// TIA Portal V15.1 export
// export: Created 2024-06-21T08:41:20.379845Z, ExportSetting WithDefaults, DisplayName Totally Integrated Automation Portal, DisplayVersion V15.1 Update 5, DisplayName TIA Portal Openness, DisplayVersion V15.1 Update 5, DisplayName SINAMICS Startdrive Advanced, DisplayVersion V15.1, DisplayName G130, G150, S120, S150, SINAMICS MV, S210, DisplayVersion V15.1, DisplayName G110M, G120, G120C, G120D, G120P, DisplayVersion V15.1, DisplayName STEP 7 Professional, DisplayVersion V15.1 Update 5, DisplayName STEP 7 Safety, DisplayVersion V15.1, DisplayName WinCC Professional, DisplayVersion V15.1 Update 5, DisplayName SIMATIC Visualization Architect, DisplayVersion V15.1
FUNCTION_BLOCK "LGBCRClockStartStop"   // FB6679, FBD
TITLE = LGBCRClockStartStop
{ S7_Optimized_Access := 'TRUE' }
VERSION : 0.1
// stored: AutoNumber false, IsIECCheckEnabled false, IsRetainMemResEnabled false, MemoryReserve 100, SetENOAutomatically False, UDAEnableTagReadback false
   VAR_INPUT
      I_DBRecieve { ExternalAccessible := 'False'; ExternalVisible := 'False'; ExternalWritable := 'False'} : "SupervisionZM";   // Receive DB - Communication with control room
      C_EnableBreaks { ExternalAccessible := 'False'; ExternalVisible := 'False'; ExternalWritable := 'False'} : Bool;   // Enable Breaks
   END_VAR
   VAR_OUTPUT
      O_Start { ExternalAccessible := 'False'; ExternalVisible := 'False'; ExternalWritable := 'False'} : Bool;   // Start production line
      O_Stop { ExternalAccessible := 'False'; ExternalVisible := 'False'; ExternalWritable := 'False'} : Bool;   // Stop production line
      O_Break { ExternalAccessible := 'False'; ExternalVisible := 'False'; ExternalWritable := 'False'} : Bool;   // Break
      O_Rotation { ExternalAccessible := 'False'; ExternalVisible := 'False'; ExternalWritable := 'False'} : Bool;   // Rotation
      O_NbrActiveShift { ExternalAccessible := 'False'; ExternalVisible := 'False'; ExternalWritable := 'False'} : Int;   // Feedback to control room
      O_NbrActiveBreak { ExternalAccessible := 'False'; ExternalVisible := 'False'; ExternalWritable := 'False'} : Int;   // Feedback to control room
      O_AlarmABCondition { ExternalAccessible := 'False'; ExternalVisible := 'False'; ExternalWritable := 'False'} : Bool;   // Alarm AB Condition
      O_AlarmA { ExternalAccessible := 'False'; ExternalVisible := 'False'; ExternalWritable := 'False'} : Bool;   // Alarm A
      O_AlarmB { ExternalAccessible := 'False'; ExternalVisible := 'False'; ExternalWritable := 'False'} : Bool;   // Alarm B
      O_AlarmC { ExternalAccessible := 'False'; ExternalVisible := 'False'; ExternalWritable := 'False'} : Bool;   // Alarm C
      O_AlarmD { ExternalAccessible := 'False'; ExternalVisible := 'False'; ExternalWritable := 'False'} : Bool;   // Alarm D
      H_AlarmWord { ExternalAccessible := 'False'; ExternalVisible := 'False'; ExternalWritable := 'False'} : DWord;   // Alarmword for WinCC
   END_VAR
   VAR_IN_OUT
      IO_Modes : "Modes";   // Modes
      H_HMI : "H_HMI";   // Animation
      H_GBCRClockStartStop : "H_GBCRClockStartStop";   // Animation
   END_VAR
   VAR
      AD_SelForce { ExternalAccessible := 'False'; ExternalVisible := 'False'; ExternalWritable := 'False'} : Bool;   // FORCE is selected in control room
      AD_SelStop { ExternalAccessible := 'False'; ExternalVisible := 'False'; ExternalWritable := 'False'} : Bool;   // STOP is selected in control room
      AD_SelRelief { ExternalAccessible := 'False'; ExternalVisible := 'False'; ExternalWritable := 'False'} : Bool;   // RELIEF is selected in control room
      DateTimePlc { ExternalAccessible := 'False'; ExternalVisible := 'False'; ExternalWritable := 'False'} : Date_And_Time;   // Date and time from Plc
      ActualTimeOfDayPlc { ExternalAccessible := 'False'; ExternalVisible := 'False'; ExternalWritable := 'False'} : Time_Of_Day;   // Actual time of day calculated by PLC
      Shift01 { ExternalAccessible := 'False'; ExternalVisible := 'False'; ExternalWritable := 'False'} : Bool;   // Shift01 active
      Shift02 { ExternalAccessible := 'False'; ExternalVisible := 'False'; ExternalWritable := 'False'} : Bool;   // Shift02 active
      Shift03 { ExternalAccessible := 'False'; ExternalVisible := 'False'; ExternalWritable := 'False'} : Bool;   // Shift03 active
      Shift04 { ExternalAccessible := 'False'; ExternalVisible := 'False'; ExternalWritable := 'False'} : Bool;   // Shift04 active
      Shift05 { ExternalAccessible := 'False'; ExternalVisible := 'False'; ExternalWritable := 'False'} : Bool;   // Shift05 active
      Shift06 { ExternalAccessible := 'False'; ExternalVisible := 'False'; ExternalWritable := 'False'} : Bool;   // Shift06 active
      Break01 { ExternalAccessible := 'False'; ExternalVisible := 'False'; ExternalWritable := 'False'} : Bool;   // Break01 active
      Break02 { ExternalAccessible := 'False'; ExternalVisible := 'False'; ExternalWritable := 'False'} : Bool;   // Break02 active
      Break03 { ExternalAccessible := 'False'; ExternalVisible := 'False'; ExternalWritable := 'False'} : Bool;   // Break03 active
      Break04 { ExternalAccessible := 'False'; ExternalVisible := 'False'; ExternalWritable := 'False'} : Bool;   // Break04 active
      Break05 { ExternalAccessible := 'False'; ExternalVisible := 'False'; ExternalWritable := 'False'} : Bool;   // Break05 active
      Break06 { ExternalAccessible := 'False'; ExternalVisible := 'False'; ExternalWritable := 'False'} : Bool;   // Break06 active
      MorningShift_RotationTime01 { ExternalAccessible := 'False'; ExternalVisible := 'False'; ExternalWritable := 'False'} : Bool;   // Rotation active
      MorningShift_RotationTime02 { ExternalAccessible := 'False'; ExternalVisible := 'False'; ExternalWritable := 'False'} : Bool;   // Rotation active
      MorningShift_RotationTime03 { ExternalAccessible := 'False'; ExternalVisible := 'False'; ExternalWritable := 'False'} : Bool;   // Rotation active
      MorningShift_RotationTime04 { ExternalAccessible := 'False'; ExternalVisible := 'False'; ExternalWritable := 'False'} : Bool;   // Rotation active
      LateShift_RotationTime01 { ExternalAccessible := 'False'; ExternalVisible := 'False'; ExternalWritable := 'False'} : Bool;   // Rotation active
      LateShift_RotationTime02 { ExternalAccessible := 'False'; ExternalVisible := 'False'; ExternalWritable := 'False'} : Bool;   // Rotation active
      LateShift_RotationTime03 { ExternalAccessible := 'False'; ExternalVisible := 'False'; ExternalWritable := 'False'} : Bool;   // Rotation active
      LateShift_RotationTime04 { ExternalAccessible := 'False'; ExternalVisible := 'False'; ExternalWritable := 'False'} : Bool;   // Rotation active
      NightShift_RotationTime01 { ExternalAccessible := 'False'; ExternalVisible := 'False'; ExternalWritable := 'False'} : Bool;   // Rotation active
      NightShift_RotationTime02 { ExternalAccessible := 'False'; ExternalVisible := 'False'; ExternalWritable := 'False'} : Bool;   // Rotation active
      NightShift_RotationTime03 { ExternalAccessible := 'False'; ExternalVisible := 'False'; ExternalWritable := 'False'} : Bool;   // Rotation active
      NightShift_RotationTime04 { ExternalAccessible := 'False'; ExternalVisible := 'False'; ExternalWritable := 'False'} : Bool;   // Rotation active
      MorningShiftDay5_RotationTime01 { ExternalAccessible := 'False'; ExternalVisible := 'False'; ExternalWritable := 'False'} : Bool;   // Rotation active
      MorningShiftDay5_RotationTime02 { ExternalAccessible := 'False'; ExternalVisible := 'False'; ExternalWritable := 'False'} : Bool;   // Rotation active
      MorningShiftDay5_RotationTime03 { ExternalAccessible := 'False'; ExternalVisible := 'False'; ExternalWritable := 'False'} : Bool;   // Rotation active
      MorningShiftDay5_RotationTime04 { ExternalAccessible := 'False'; ExternalVisible := 'False'; ExternalWritable := 'False'} : Bool;   // Rotation active
      LateShiftDay5_RotationTime01 { ExternalAccessible := 'False'; ExternalVisible := 'False'; ExternalWritable := 'False'} : Bool;   // Rotation active
      LateShiftDay5_RotationTime02 { ExternalAccessible := 'False'; ExternalVisible := 'False'; ExternalWritable := 'False'} : Bool;   // Rotation active
      LateShiftDay5_RotationTime03 { ExternalAccessible := 'False'; ExternalVisible := 'False'; ExternalWritable := 'False'} : Bool;   // Rotation active
      LateShiftDay5_RotationTime04 { ExternalAccessible := 'False'; ExternalVisible := 'False'; ExternalWritable := 'False'} : Bool;   // Rotation active
      NightShiftDay5_RotationTime01 { ExternalAccessible := 'False'; ExternalVisible := 'False'; ExternalWritable := 'False'} : Bool;   // Rotation active
      NightShiftDay5_RotationTime02 { ExternalAccessible := 'False'; ExternalVisible := 'False'; ExternalWritable := 'False'} : Bool;   // Rotation active
      NightShiftDay5_RotationTime03 { ExternalAccessible := 'False'; ExternalVisible := 'False'; ExternalWritable := 'False'} : Bool;   // Rotation active
      NightShiftDay5_RotationTime04 { ExternalAccessible := 'False'; ExternalVisible := 'False'; ExternalWritable := 'False'} : Bool;   // Rotation active
      ShiftActive { ExternalAccessible := 'False'; ExternalVisible := 'False'; ExternalWritable := 'False'} : Bool;   // Shift active
      BreakActive { ExternalAccessible := 'False'; ExternalVisible := 'False'; ExternalWritable := 'False'} : Bool;   // Break active
      RotationActive { ExternalAccessible := 'False'; ExternalVisible := 'False'; ExternalWritable := 'False'} : Bool;   // Rotation active
      Production { ExternalAccessible := 'False'; ExternalVisible := 'False'; ExternalWritable := 'False'} : Bool;   // In production, production line can RUN
      Start { ExternalAccessible := 'False'; ExternalVisible := 'False'; ExternalWritable := 'False'} : Bool;   // Start production line
      Stop { ExternalAccessible := 'False'; ExternalVisible := 'False'; ExternalWritable := 'False'} : Bool;   // Stop production line
      NbrActiveShift { ExternalAccessible := 'False'; ExternalVisible := 'False'; ExternalWritable := 'False'} : Int;   // Feedback to control room
      NbrActiveBreak { ExternalAccessible := 'False'; ExternalVisible := 'False'; ExternalWritable := 'False'} : Int;   // Feedback to control room
      AlarmA { ExternalAccessible := 'False'; ExternalVisible := 'False'; ExternalWritable := 'False'} : Bool;   // Alarm A
      AlarmB { ExternalAccessible := 'False'; ExternalVisible := 'False'; ExternalWritable := 'False'} : Bool;   // Alarm B
      AlarmC { ExternalAccessible := 'False'; ExternalVisible := 'False'; ExternalWritable := 'False'} : Bool;   // Alarm C
      AlarmD { ExternalAccessible := 'False'; ExternalVisible := 'False'; ExternalWritable := 'False'} : Bool;   // Alarm D
      AlarmABCondition { ExternalAccessible := 'False'; ExternalVisible := 'False'; ExternalWritable := 'False'} : Bool;   // Alarm AB Condition
      RotationTime { ExternalAccessible := 'False'; ExternalVisible := 'False'; ExternalWritable := 'False'} : Time_Of_Day;   // Rotation Time
      MorningShift_RotationTime01_End { ExternalAccessible := 'False'; ExternalVisible := 'False'; ExternalWritable := 'False'} : Time_Of_Day;   // Rotation End Time
      MorningShift_RotationTime02_End { ExternalAccessible := 'False'; ExternalVisible := 'False'; ExternalWritable := 'False'} : Time_Of_Day;   // Rotation End Time
      MorningShift_RotationTime03_End { ExternalAccessible := 'False'; ExternalVisible := 'False'; ExternalWritable := 'False'} : Time_Of_Day;   // Rotation End Time
      MorningShift_RotationTime04_End { ExternalAccessible := 'False'; ExternalVisible := 'False'; ExternalWritable := 'False'} : Time_Of_Day;   // Rotation End Time
      LateShift_RotationTime01_End { ExternalAccessible := 'False'; ExternalVisible := 'False'; ExternalWritable := 'False'} : Time_Of_Day;   // Rotation End Time
      LateShift_RotationTime02_End { ExternalAccessible := 'False'; ExternalVisible := 'False'; ExternalWritable := 'False'} : Time_Of_Day;   // Rotation End Time
      LateShift_RotationTime03_End { ExternalAccessible := 'False'; ExternalVisible := 'False'; ExternalWritable := 'False'} : Time_Of_Day;   // Rotation End Time
      LateShift_RotationTime04_End { ExternalAccessible := 'False'; ExternalVisible := 'False'; ExternalWritable := 'False'} : Time_Of_Day;   // Rotation End Time
      NightShift_RotationTime01_End { ExternalAccessible := 'False'; ExternalVisible := 'False'; ExternalWritable := 'False'} : Time_Of_Day;   // Rotation End Time
      NightShift_RotationTime02_End { ExternalAccessible := 'False'; ExternalVisible := 'False'; ExternalWritable := 'False'} : Time_Of_Day;   // Rotation End Time
      NightShift_RotationTime03_End { ExternalAccessible := 'False'; ExternalVisible := 'False'; ExternalWritable := 'False'} : Time_Of_Day;   // Rotation End Time
      NightShift_RotationTime04_End { ExternalAccessible := 'False'; ExternalVisible := 'False'; ExternalWritable := 'False'} : Time_Of_Day;   // Rotation End Time
      MorningShiftDay5_RotationTime01_End { ExternalAccessible := 'False'; ExternalVisible := 'False'; ExternalWritable := 'False'} : Time_Of_Day;   // Rotation End Time
      MorningShiftDay5_RotationTime02_End { ExternalAccessible := 'False'; ExternalVisible := 'False'; ExternalWritable := 'False'} : Time_Of_Day;   // Rotation End Time
      MorningShiftDay5_RotationTime03_End { ExternalAccessible := 'False'; ExternalVisible := 'False'; ExternalWritable := 'False'} : Time_Of_Day;   // Rotation End Time
      MorningShiftDay5_RotationTime04_End { ExternalAccessible := 'False'; ExternalVisible := 'False'; ExternalWritable := 'False'} : Time_Of_Day;   // Rotation End Time
      LateShiftDay5_RotationTime01_End { ExternalAccessible := 'False'; ExternalVisible := 'False'; ExternalWritable := 'False'} : Time_Of_Day;   // Rotation End Time
      LateShiftDay5_RotationTime02_End { ExternalAccessible := 'False'; ExternalVisible := 'False'; ExternalWritable := 'False'} : Time_Of_Day;   // Rotation End Time
      LateShiftDay5_RotationTime03_End { ExternalAccessible := 'False'; ExternalVisible := 'False'; ExternalWritable := 'False'} : Time_Of_Day;   // Rotation End Time
      LateShiftDay5_RotationTime04_End { ExternalAccessible := 'False'; ExternalVisible := 'False'; ExternalWritable := 'False'} : Time_Of_Day;   // Rotation End Time
      NightShiftDay5_RotationTime01_End { ExternalAccessible := 'False'; ExternalVisible := 'False'; ExternalWritable := 'False'} : Time_Of_Day;   // Rotation End Time
      NightShiftDay5_RotationTime02_End { ExternalAccessible := 'False'; ExternalVisible := 'False'; ExternalWritable := 'False'} : Time_Of_Day;   // Rotation End Time
      NightShiftDay5_RotationTime03_End { ExternalAccessible := 'False'; ExternalVisible := 'False'; ExternalWritable := 'False'} : Time_Of_Day;   // Rotation End Time
      NightShiftDay5_RotationTime04_End { ExternalAccessible := 'False'; ExternalVisible := 'False'; ExternalWritable := 'False'} : Time_Of_Day;   // Rotation End Time
      HMICmdCR { ExternalAccessible := 'False'; ExternalVisible := 'False'; ExternalWritable := 'False'} : Struct   // Temp / HMI Commands control room
         SelForce { ExternalAccessible := 'False'; ExternalVisible := 'False'; ExternalWritable := 'False'} : Bool;   // FORCE is selected in control room
         SelStop { ExternalAccessible := 'False'; ExternalVisible := 'False'; ExternalWritable := 'False'} : Bool;   // STOP is selected in control room
         SelRelief { ExternalAccessible := 'False'; ExternalVisible := 'False'; ExternalWritable := 'False'} : Bool;   // RELIEF is selected in control room
         Spare3 { ExternalAccessible := 'False'; ExternalVisible := 'False'; ExternalWritable := 'False'} : Bool;   // Spare
         Spare4 { ExternalAccessible := 'False'; ExternalVisible := 'False'; ExternalWritable := 'False'} : Bool;   // Spare
         Spare5 { ExternalAccessible := 'False'; ExternalVisible := 'False'; ExternalWritable := 'False'} : Bool;   // Spare
         Spare6 { ExternalAccessible := 'False'; ExternalVisible := 'False'; ExternalWritable := 'False'} : Bool;   // Spare
         Spare7 { ExternalAccessible := 'False'; ExternalVisible := 'False'; ExternalWritable := 'False'} : Bool;   // Spare
         Spare8 { ExternalAccessible := 'False'; ExternalVisible := 'False'; ExternalWritable := 'False'} : Bool;   // Spare
         Spare9 { ExternalAccessible := 'False'; ExternalVisible := 'False'; ExternalWritable := 'False'} : Bool;   // Spare
         Spare10 { ExternalAccessible := 'False'; ExternalVisible := 'False'; ExternalWritable := 'False'} : Bool;   // Spare
         Spare11 { ExternalAccessible := 'False'; ExternalVisible := 'False'; ExternalWritable := 'False'} : Bool;   // Spare
         Spare12 { ExternalAccessible := 'False'; ExternalVisible := 'False'; ExternalWritable := 'False'} : Bool;   // Spare
         Spare13 { ExternalAccessible := 'False'; ExternalVisible := 'False'; ExternalWritable := 'False'} : Bool;   // Spare
         Spare14 { ExternalAccessible := 'False'; ExternalVisible := 'False'; ExternalWritable := 'False'} : Bool;   // Spare
         Spare15 { ExternalAccessible := 'False'; ExternalVisible := 'False'; ExternalWritable := 'False'} : Bool;   // Spare
         Spare16 { ExternalAccessible := 'False'; ExternalVisible := 'False'; ExternalWritable := 'False'} : Bool;   // Spare
         Spare17 { ExternalAccessible := 'False'; ExternalVisible := 'False'; ExternalWritable := 'False'} : Bool;   // Spare
         Spare18 { ExternalAccessible := 'False'; ExternalVisible := 'False'; ExternalWritable := 'False'} : Bool;   // Spare
         Spare19 { ExternalAccessible := 'False'; ExternalVisible := 'False'; ExternalWritable := 'False'} : Bool;   // Spare
         Spare20 { ExternalAccessible := 'False'; ExternalVisible := 'False'; ExternalWritable := 'False'} : Bool;   // Spare
         Spare21 { ExternalAccessible := 'False'; ExternalVisible := 'False'; ExternalWritable := 'False'} : Bool;   // Spare
         Spare22 { ExternalAccessible := 'False'; ExternalVisible := 'False'; ExternalWritable := 'False'} : Bool;   // Spare
         Spare23 { ExternalAccessible := 'False'; ExternalVisible := 'False'; ExternalWritable := 'False'} : Bool;   // Spare
         Spare24 { ExternalAccessible := 'False'; ExternalVisible := 'False'; ExternalWritable := 'False'} : Bool;   // Spare
         Spare25 { ExternalAccessible := 'False'; ExternalVisible := 'False'; ExternalWritable := 'False'} : Bool;   // Spare
         Spare26 { ExternalAccessible := 'False'; ExternalVisible := 'False'; ExternalWritable := 'False'} : Bool;   // Spare
         Spare27 { ExternalAccessible := 'False'; ExternalVisible := 'False'; ExternalWritable := 'False'} : Bool;   // Spare
         Spare28 { ExternalAccessible := 'False'; ExternalVisible := 'False'; ExternalWritable := 'False'} : Bool;   // Spare
         Spare29 { ExternalAccessible := 'False'; ExternalVisible := 'False'; ExternalWritable := 'False'} : Bool;   // Spare
         Spare30 { ExternalAccessible := 'False'; ExternalVisible := 'False'; ExternalWritable := 'False'} : Bool;   // Spare
         Spare31 { ExternalAccessible := 'False'; ExternalVisible := 'False'; ExternalWritable := 'False'} : Bool;   // Spare
      END_STRUCT;
      HMICmd { ExternalAccessible := 'False'; ExternalVisible := 'False'; ExternalWritable := 'False'} : Struct   // HMI Commands
         MorningShift_RotationTime01_Active { ExternalAccessible := 'False'; ExternalVisible := 'False'; ExternalWritable := 'False'} : Bool;   // Rotation time active
         MorningShift_RotationTime02_Active { ExternalAccessible := 'False'; ExternalVisible := 'False'; ExternalWritable := 'False'} : Bool;   // Rotation time active
         MorningShift_RotationTime03_Active { ExternalAccessible := 'False'; ExternalVisible := 'False'; ExternalWritable := 'False'} : Bool;   // Rotation time active
         MorningShift_RotationTime04_Active { ExternalAccessible := 'False'; ExternalVisible := 'False'; ExternalWritable := 'False'} : Bool;   // Rotation time active
         LateShift_RotationTime01_Active { ExternalAccessible := 'False'; ExternalVisible := 'False'; ExternalWritable := 'False'} : Bool;   // Rotation time active
         LateShift_RotationTime02_Active { ExternalAccessible := 'False'; ExternalVisible := 'False'; ExternalWritable := 'False'} : Bool;   // Rotation time active
         LateShift_RotationTime03_Active { ExternalAccessible := 'False'; ExternalVisible := 'False'; ExternalWritable := 'False'} : Bool;   // Rotation time active
         LateShift_RotationTime04_Active { ExternalAccessible := 'False'; ExternalVisible := 'False'; ExternalWritable := 'False'} : Bool;   // Rotation time active
         NightShift_RotationTime01_Active { ExternalAccessible := 'False'; ExternalVisible := 'False'; ExternalWritable := 'False'} : Bool;   // Rotation time active
         NightShift_RotationTime02_Active { ExternalAccessible := 'False'; ExternalVisible := 'False'; ExternalWritable := 'False'} : Bool;   // Rotation time active
         NightShift_RotationTime03_Active { ExternalAccessible := 'False'; ExternalVisible := 'False'; ExternalWritable := 'False'} : Bool;   // Rotation time active
         NightShift_RotationTime04_Active { ExternalAccessible := 'False'; ExternalVisible := 'False'; ExternalWritable := 'False'} : Bool;   // Rotation time active
         MorningShiftDay5_RotationTime01_Active { ExternalAccessible := 'False'; ExternalVisible := 'False'; ExternalWritable := 'False'} : Bool;   // Rotation time active
         MorningShiftDay5_RotationTime02_Active { ExternalAccessible := 'False'; ExternalVisible := 'False'; ExternalWritable := 'False'} : Bool;   // Rotation time active
         MorningShiftDay5_RotationTime03_Active { ExternalAccessible := 'False'; ExternalVisible := 'False'; ExternalWritable := 'False'} : Bool;   // Rotation time active
         MorningShiftDay5_RotationTime04_Active { ExternalAccessible := 'False'; ExternalVisible := 'False'; ExternalWritable := 'False'} : Bool;   // Rotation time active
         LateShiftDay5_RotationTime01_Active { ExternalAccessible := 'False'; ExternalVisible := 'False'; ExternalWritable := 'False'} : Bool;   // Rotation time active
         LateShiftDay5_RotationTime02_Active { ExternalAccessible := 'False'; ExternalVisible := 'False'; ExternalWritable := 'False'} : Bool;   // Rotation time active
         LateShiftDay5_RotationTime03_Active { ExternalAccessible := 'False'; ExternalVisible := 'False'; ExternalWritable := 'False'} : Bool;   // Rotation time active
         LateShiftDay5_RotationTime04_Active { ExternalAccessible := 'False'; ExternalVisible := 'False'; ExternalWritable := 'False'} : Bool;   // Rotation time active
         NightShiftDay5_RotationTime01_Active { ExternalAccessible := 'False'; ExternalVisible := 'False'; ExternalWritable := 'False'} : Bool;   // Rotation time active
         NightShiftDay5_RotationTime02_Active { ExternalAccessible := 'False'; ExternalVisible := 'False'; ExternalWritable := 'False'} : Bool;   // Rotation time active
         NightShiftDay5_RotationTime03_Active { ExternalAccessible := 'False'; ExternalVisible := 'False'; ExternalWritable := 'False'} : Bool;   // Rotation time active
         NightShiftDay5_RotationTime04_Active { ExternalAccessible := 'False'; ExternalVisible := 'False'; ExternalWritable := 'False'} : Bool;   // Rotation time active
      END_STRUCT;
   END_VAR
   VAR_TEMP
      TReadStatus : Int;   // Integer used store the status of the clock read
      TempTime : Time_Of_Day;
   END_VAR
   VAR_TEMP   // added for the SCL form of the ladder/FBD networks
      _w1 : Bool;
   END_VAR
BEGIN

REGION Network 1: **** 1 - Inputs **** HMI Commands / **** 1 - Inputs **** HMI Commands !!! Control room !!!
   // HMI Commands
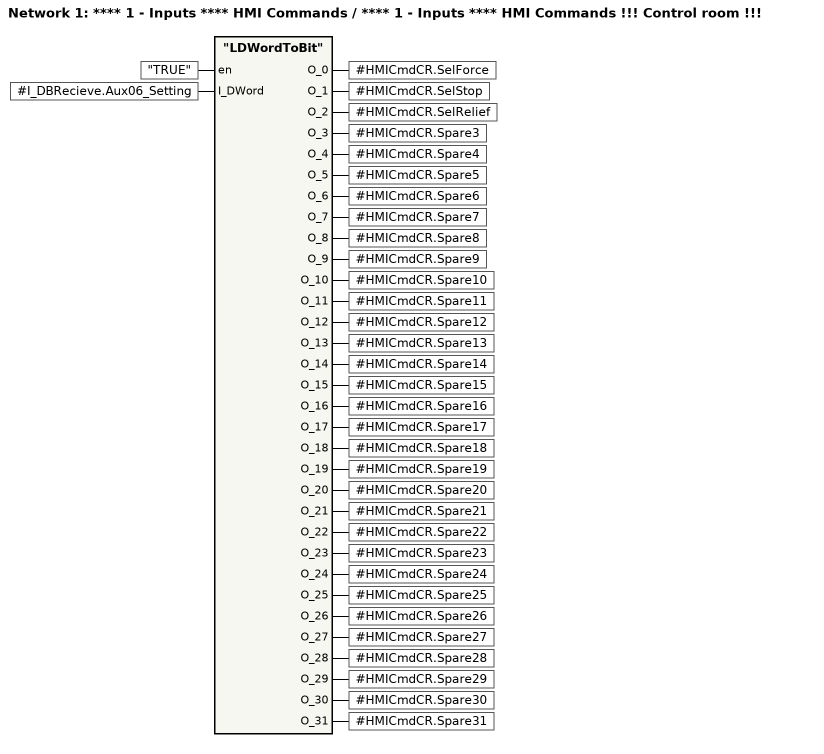
   IF "TRUE" THEN
       "LDWordToBit"(I_DWord := #I_DBRecieve.Aux06_Setting,
                     O_0 => #HMICmdCR.SelForce,
                     O_1 => #HMICmdCR.SelStop,
                     O_2 => #HMICmdCR.SelRelief,
                     O_3 => #HMICmdCR.Spare3,
                     O_4 => #HMICmdCR.Spare4,
                     O_5 => #HMICmdCR.Spare5,
                     O_6 => #HMICmdCR.Spare6,
                     O_7 => #HMICmdCR.Spare7,
                     O_8 => #HMICmdCR.Spare8,
                     O_9 => #HMICmdCR.Spare9,
                     O_10 => #HMICmdCR.Spare10,
                     O_11 => #HMICmdCR.Spare11,
                     O_12 => #HMICmdCR.Spare12,
                     O_13 => #HMICmdCR.Spare13,
                     O_14 => #HMICmdCR.Spare14,
                     O_15 => #HMICmdCR.Spare15,
                     O_16 => #HMICmdCR.Spare16,
                     O_17 => #HMICmdCR.Spare17,
                     O_18 => #HMICmdCR.Spare18,
                     O_19 => #HMICmdCR.Spare19,
                     O_20 => #HMICmdCR.Spare20,
                     O_21 => #HMICmdCR.Spare21,
                     O_22 => #HMICmdCR.Spare22,
                     O_23 => #HMICmdCR.Spare23,
                     O_24 => #HMICmdCR.Spare24,
                     O_25 => #HMICmdCR.Spare25,
                     O_26 => #HMICmdCR.Spare26,
                     O_27 => #HMICmdCR.Spare27,
                     O_28 => #HMICmdCR.Spare28,
                     O_29 => #HMICmdCR.Spare29,
                     O_30 => #HMICmdCR.Spare30,
                     O_31 => #HMICmdCR.Spare31);
   END_IF;
END_REGION

REGION Network 2: **** 1 - Inputs **** HMI Commands
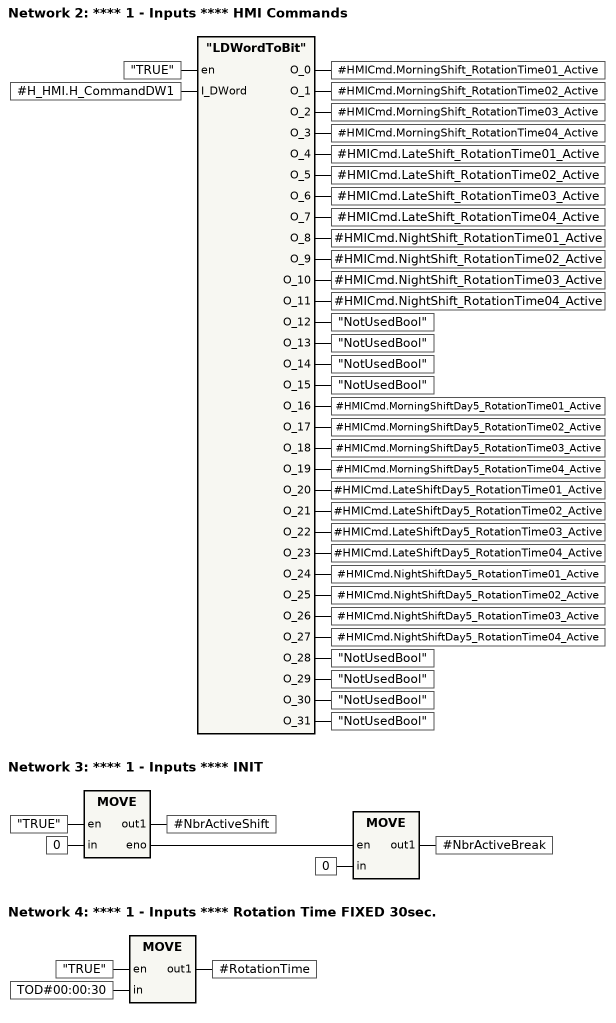
   IF "TRUE" THEN
       "LDWordToBit"(I_DWord := #H_HMI.H_CommandDW1,
                     O_0 => #HMICmd.MorningShift_RotationTime01_Active,
                     O_1 => #HMICmd.MorningShift_RotationTime02_Active,
                     O_2 => #HMICmd.MorningShift_RotationTime03_Active,
                     O_3 => #HMICmd.MorningShift_RotationTime04_Active,
                     O_4 => #HMICmd.LateShift_RotationTime01_Active,
                     O_5 => #HMICmd.LateShift_RotationTime02_Active,
                     O_6 => #HMICmd.LateShift_RotationTime03_Active,
                     O_7 => #HMICmd.LateShift_RotationTime04_Active,
                     O_8 => #HMICmd.NightShift_RotationTime01_Active,
                     O_9 => #HMICmd.NightShift_RotationTime02_Active,
                     O_10 => #HMICmd.NightShift_RotationTime03_Active,
                     O_11 => #HMICmd.NightShift_RotationTime04_Active,
                     O_12 => "NotUsedBool",
                     O_13 => "NotUsedBool",
                     O_14 => "NotUsedBool",
                     O_15 => "NotUsedBool",
                     O_16 => #HMICmd.MorningShiftDay5_RotationTime01_Active,
                     O_17 => #HMICmd.MorningShiftDay5_RotationTime02_Active,
                     O_18 => #HMICmd.MorningShiftDay5_RotationTime03_Active,
                     O_19 => #HMICmd.MorningShiftDay5_RotationTime04_Active,
                     O_20 => #HMICmd.LateShiftDay5_RotationTime01_Active,
                     O_21 => #HMICmd.LateShiftDay5_RotationTime02_Active,
                     O_22 => #HMICmd.LateShiftDay5_RotationTime03_Active,
                     O_23 => #HMICmd.LateShiftDay5_RotationTime04_Active,
                     O_24 => #HMICmd.NightShiftDay5_RotationTime01_Active,
                     O_25 => #HMICmd.NightShiftDay5_RotationTime02_Active,
                     O_26 => #HMICmd.NightShiftDay5_RotationTime03_Active,
                     O_27 => #HMICmd.NightShiftDay5_RotationTime04_Active,
                     O_28 => "NotUsedBool",
                     O_29 => "NotUsedBool",
                     O_30 => "NotUsedBool",
                     O_31 => "NotUsedBool");
   END_IF;
END_REGION

REGION Network 3: **** 1 - Inputs **** INIT
   IF "TRUE" THEN
       #NbrActiveShift := 0;
       #NbrActiveBreak := 0;
   END_IF;
END_REGION

REGION Network 4: **** 1 - Inputs **** Rotation Time FIXED 30sec.
   IF "TRUE" THEN #RotationTime := TOD#00:00:30; END_IF;
END_REGION

REGION Network 5: **** 1 - Inputs **** Rotation End Time Morning Shift
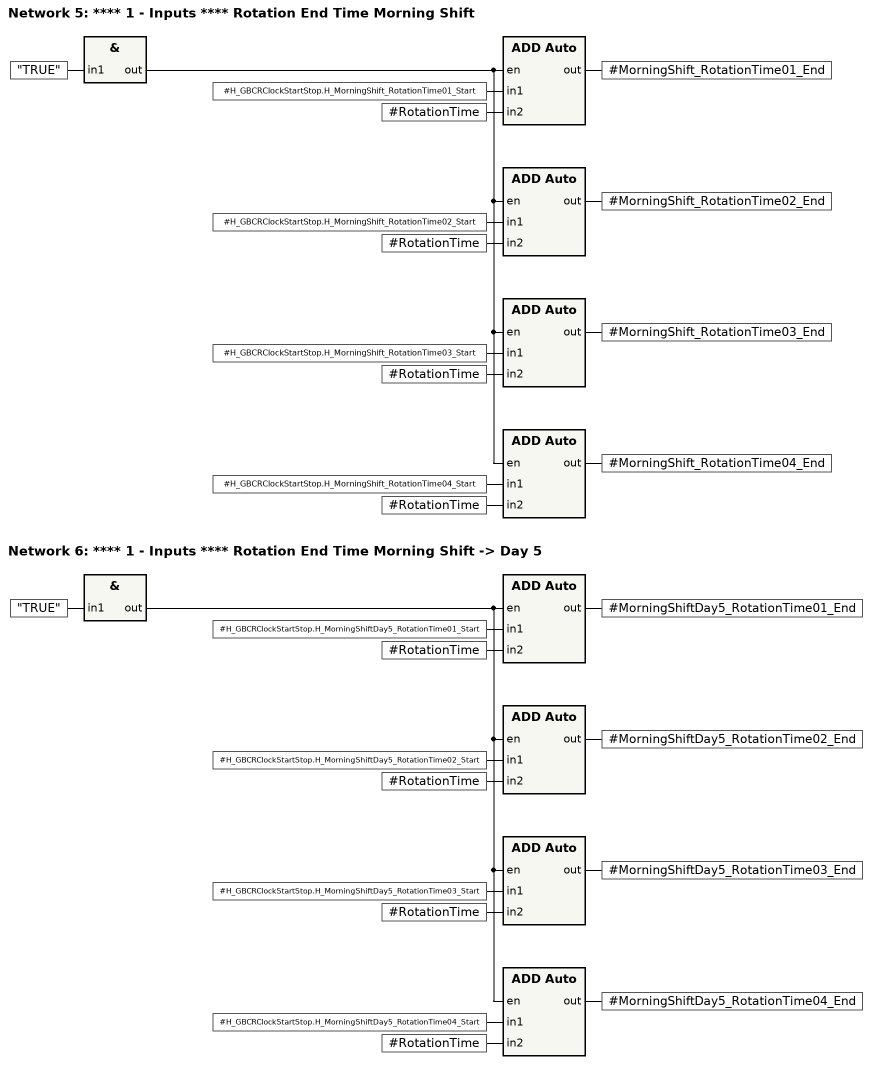
   IF "TRUE" THEN
       #MorningShift_RotationTime01_End := #H_GBCRClockStartStop.H_MorningShift_RotationTime01_Start + #RotationTime;
       #MorningShift_RotationTime02_End := #H_GBCRClockStartStop.H_MorningShift_RotationTime02_Start + #RotationTime;
       #MorningShift_RotationTime03_End := #H_GBCRClockStartStop.H_MorningShift_RotationTime03_Start + #RotationTime;
       #MorningShift_RotationTime04_End := #H_GBCRClockStartStop.H_MorningShift_RotationTime04_Start + #RotationTime;
   END_IF;
END_REGION

REGION Network 6: **** 1 - Inputs **** Rotation End Time Morning Shift -> Day 5
   IF "TRUE" THEN
       #MorningShiftDay5_RotationTime01_End := #H_GBCRClockStartStop.H_MorningShiftDay5_RotationTime01_Start + #RotationTime;
       #MorningShiftDay5_RotationTime02_End := #H_GBCRClockStartStop.H_MorningShiftDay5_RotationTime02_Start + #RotationTime;
       #MorningShiftDay5_RotationTime03_End := #H_GBCRClockStartStop.H_MorningShiftDay5_RotationTime03_Start + #RotationTime;
       #MorningShiftDay5_RotationTime04_End := #H_GBCRClockStartStop.H_MorningShiftDay5_RotationTime04_Start + #RotationTime;
   END_IF;
END_REGION

REGION Network 7: **** 1 - Inputs **** Rotation End Time Late Shift
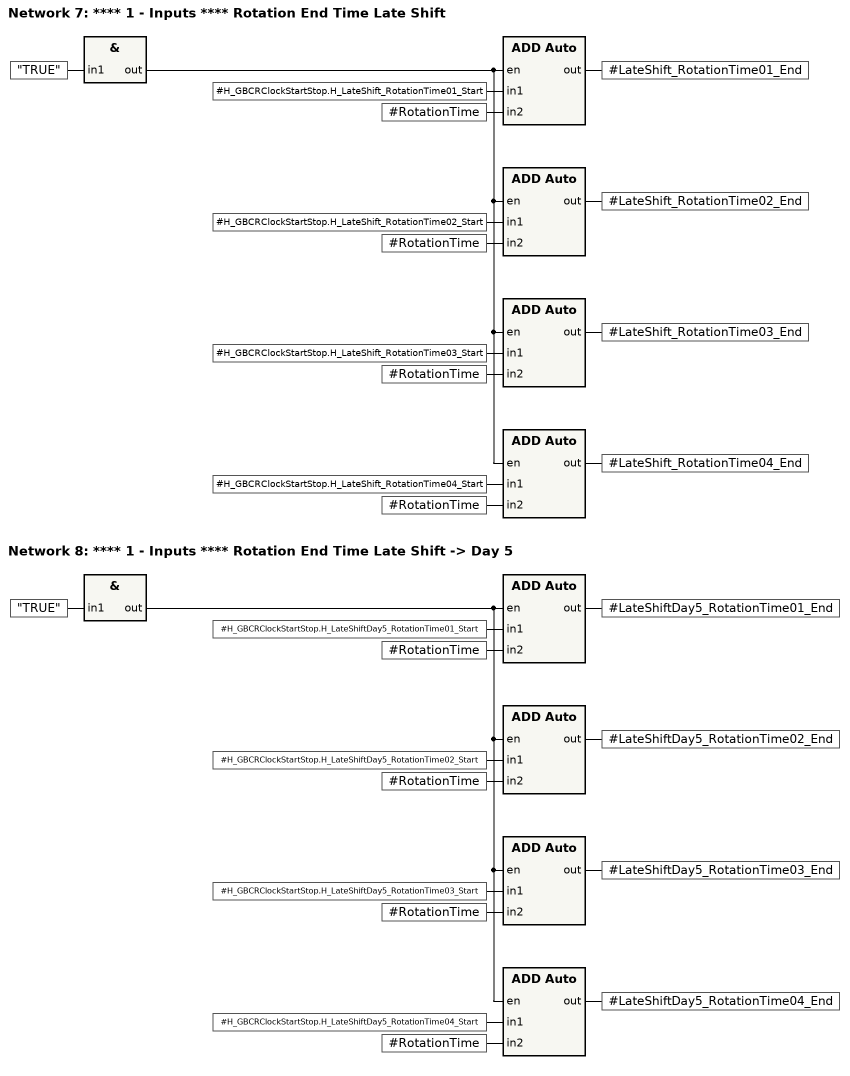
   IF "TRUE" THEN
       #LateShift_RotationTime01_End := #H_GBCRClockStartStop.H_LateShift_RotationTime01_Start + #RotationTime;
       #LateShift_RotationTime02_End := #H_GBCRClockStartStop.H_LateShift_RotationTime02_Start + #RotationTime;
       #LateShift_RotationTime03_End := #H_GBCRClockStartStop.H_LateShift_RotationTime03_Start + #RotationTime;
       #LateShift_RotationTime04_End := #H_GBCRClockStartStop.H_LateShift_RotationTime04_Start + #RotationTime;
   END_IF;
END_REGION

REGION Network 8: **** 1 - Inputs **** Rotation End Time Late Shift -> Day 5
   IF "TRUE" THEN
       #LateShiftDay5_RotationTime01_End := #H_GBCRClockStartStop.H_LateShiftDay5_RotationTime01_Start + #RotationTime;
       #LateShiftDay5_RotationTime02_End := #H_GBCRClockStartStop.H_LateShiftDay5_RotationTime02_Start + #RotationTime;
       #LateShiftDay5_RotationTime03_End := #H_GBCRClockStartStop.H_LateShiftDay5_RotationTime03_Start + #RotationTime;
       #LateShiftDay5_RotationTime04_End := #H_GBCRClockStartStop.H_LateShiftDay5_RotationTime04_Start + #RotationTime;
   END_IF;
END_REGION

REGION Network 9: **** 1 - Inputs **** Rotation End Time Night Shift
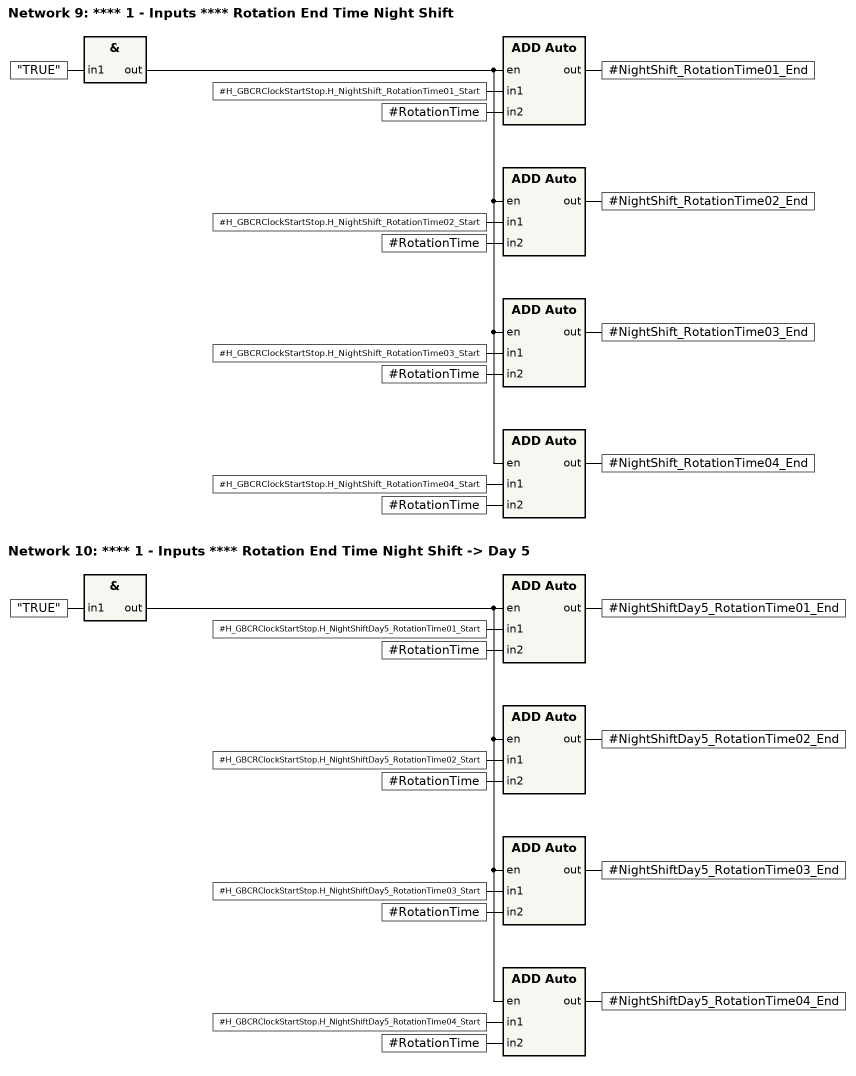
   IF "TRUE" THEN
       #NightShift_RotationTime01_End := #H_GBCRClockStartStop.H_NightShift_RotationTime01_Start + #RotationTime;
       #NightShift_RotationTime02_End := #H_GBCRClockStartStop.H_NightShift_RotationTime02_Start + #RotationTime;
       #NightShift_RotationTime03_End := #H_GBCRClockStartStop.H_NightShift_RotationTime03_Start + #RotationTime;
       #NightShift_RotationTime04_End := #H_GBCRClockStartStop.H_NightShift_RotationTime04_Start + #RotationTime;
   END_IF;
END_REGION

REGION Network 10: **** 1 - Inputs **** Rotation End Time Night Shift -> Day 5
   IF "TRUE" THEN
       #NightShiftDay5_RotationTime01_End := #H_GBCRClockStartStop.H_NightShiftDay5_RotationTime01_Start + #RotationTime;
       #NightShiftDay5_RotationTime02_End := #H_GBCRClockStartStop.H_NightShiftDay5_RotationTime02_Start + #RotationTime;
       #NightShiftDay5_RotationTime03_End := #H_GBCRClockStartStop.H_NightShiftDay5_RotationTime03_Start + #RotationTime;
       #NightShiftDay5_RotationTime04_End := #H_GBCRClockStartStop.H_NightShiftDay5_RotationTime04_Start + #RotationTime;
   END_IF;
END_REGION

REGION Network 11: **** 1 - Inputs **** Rotation End Time Night Shift -> If start time > then 23:59:29
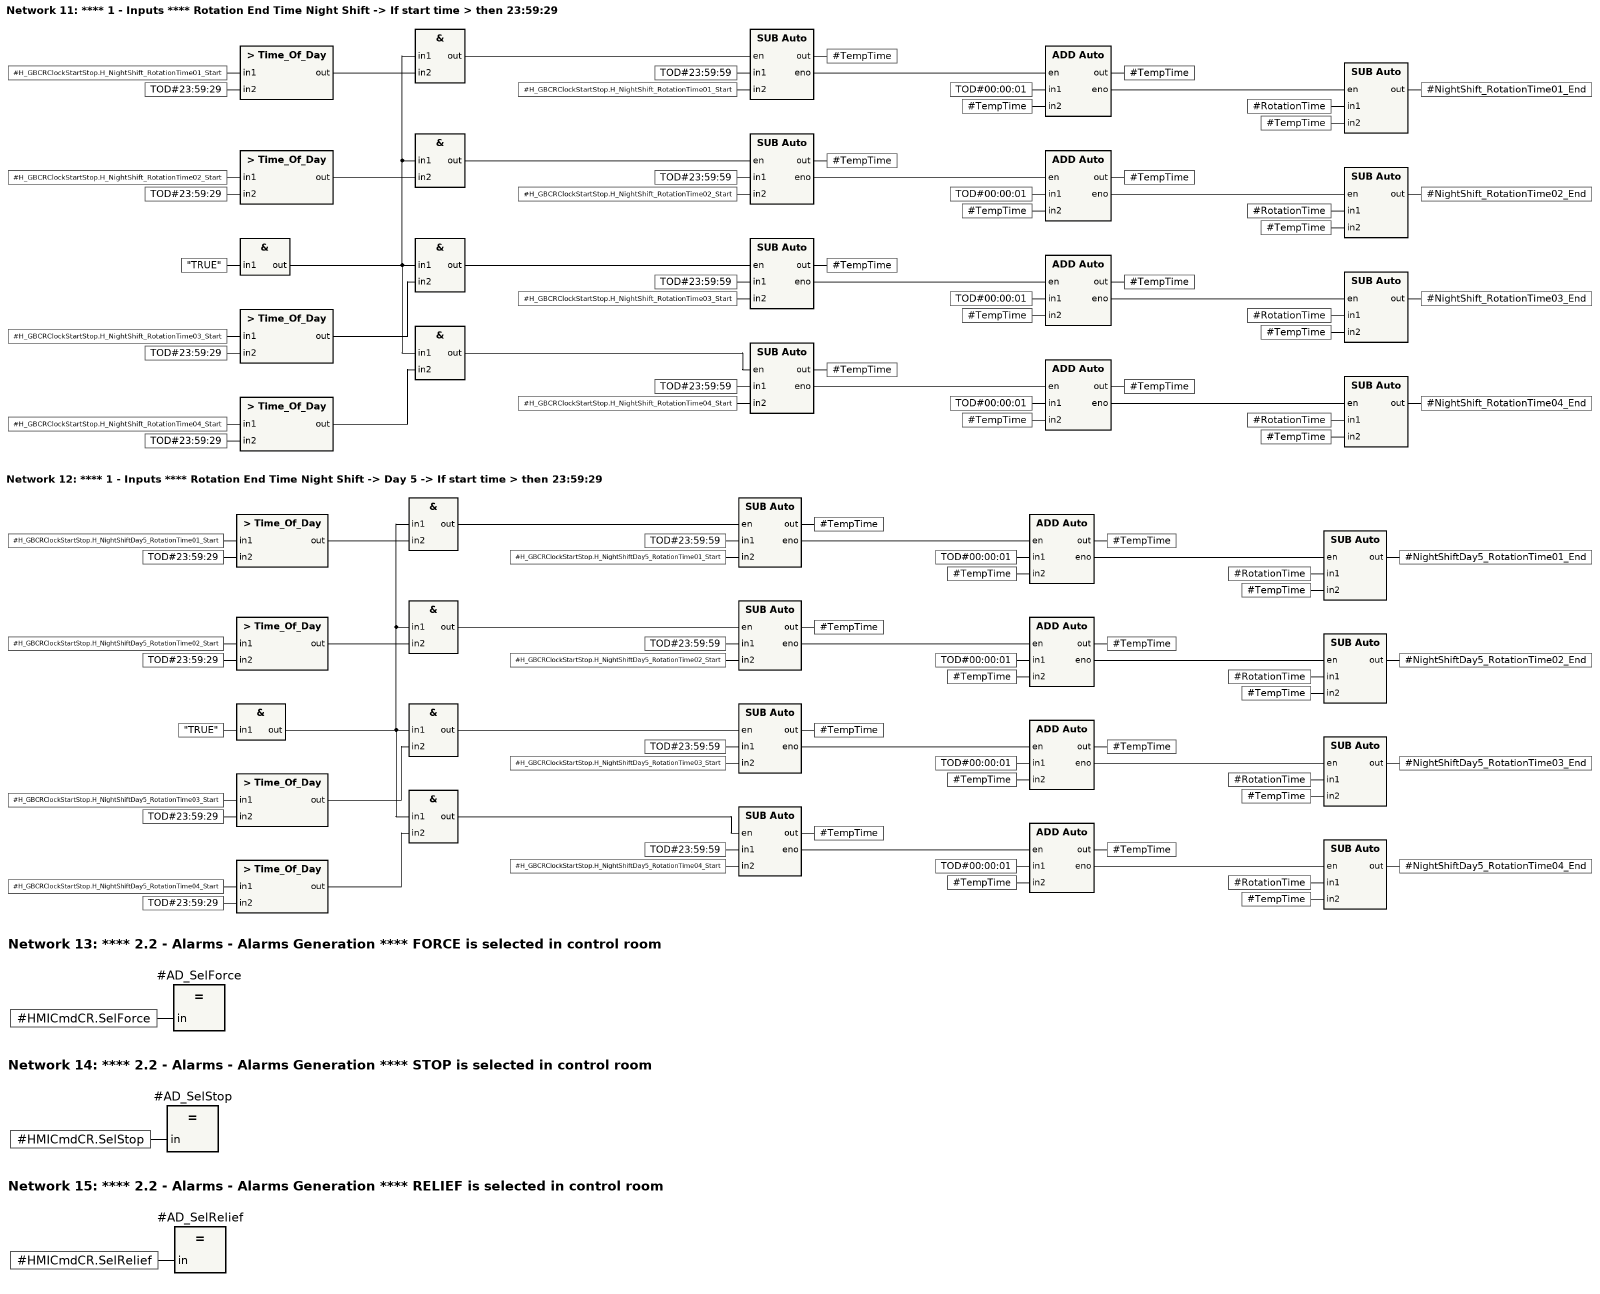
   IF "TRUE" AND (#H_GBCRClockStartStop.H_NightShift_RotationTime01_Start > TOD#23:59:29) THEN
       #TempTime := TOD#23:59:59 - #H_GBCRClockStartStop.H_NightShift_RotationTime01_Start;
       #TempTime := TOD#00:00:01 + #TempTime;
       #NightShift_RotationTime01_End := #RotationTime - #TempTime;
   END_IF;
   IF "TRUE" AND (#H_GBCRClockStartStop.H_NightShift_RotationTime02_Start > TOD#23:59:29) THEN
       #TempTime := TOD#23:59:59 - #H_GBCRClockStartStop.H_NightShift_RotationTime02_Start;
       #TempTime := TOD#00:00:01 + #TempTime;
       #NightShift_RotationTime02_End := #RotationTime - #TempTime;
   END_IF;
   IF "TRUE" AND (#H_GBCRClockStartStop.H_NightShift_RotationTime03_Start > TOD#23:59:29) THEN
       #TempTime := TOD#23:59:59 - #H_GBCRClockStartStop.H_NightShift_RotationTime03_Start;
       #TempTime := TOD#00:00:01 + #TempTime;
       #NightShift_RotationTime03_End := #RotationTime - #TempTime;
   END_IF;
   IF "TRUE" AND (#H_GBCRClockStartStop.H_NightShift_RotationTime04_Start > TOD#23:59:29) THEN
       #TempTime := TOD#23:59:59 - #H_GBCRClockStartStop.H_NightShift_RotationTime04_Start;
       #TempTime := TOD#00:00:01 + #TempTime;
       #NightShift_RotationTime04_End := #RotationTime - #TempTime;
   END_IF;
END_REGION

REGION Network 12: **** 1 - Inputs **** Rotation End Time Night Shift -> Day 5 -> If start time > then 23:59:29
   IF "TRUE" AND (#H_GBCRClockStartStop.H_NightShiftDay5_RotationTime01_Start > TOD#23:59:29) THEN
       #TempTime := TOD#23:59:59 - #H_GBCRClockStartStop.H_NightShiftDay5_RotationTime01_Start;
       #TempTime := TOD#00:00:01 + #TempTime;
       #NightShiftDay5_RotationTime01_End := #RotationTime - #TempTime;
   END_IF;
   IF "TRUE" AND (#H_GBCRClockStartStop.H_NightShiftDay5_RotationTime02_Start > TOD#23:59:29) THEN
       #TempTime := TOD#23:59:59 - #H_GBCRClockStartStop.H_NightShiftDay5_RotationTime02_Start;
       #TempTime := TOD#00:00:01 + #TempTime;
       #NightShiftDay5_RotationTime02_End := #RotationTime - #TempTime;
   END_IF;
   IF "TRUE" AND (#H_GBCRClockStartStop.H_NightShiftDay5_RotationTime03_Start > TOD#23:59:29) THEN
       #TempTime := TOD#23:59:59 - #H_GBCRClockStartStop.H_NightShiftDay5_RotationTime03_Start;
       #TempTime := TOD#00:00:01 + #TempTime;
       #NightShiftDay5_RotationTime03_End := #RotationTime - #TempTime;
   END_IF;
   IF "TRUE" AND (#H_GBCRClockStartStop.H_NightShiftDay5_RotationTime04_Start > TOD#23:59:29) THEN
       #TempTime := TOD#23:59:59 - #H_GBCRClockStartStop.H_NightShiftDay5_RotationTime04_Start;
       #TempTime := TOD#00:00:01 + #TempTime;
       #NightShiftDay5_RotationTime04_End := #RotationTime - #TempTime;
   END_IF;
END_REGION

REGION Network 13: **** 2.2 - Alarms - Alarms Generation **** FORCE is selected in control room
   #AD_SelForce := #HMICmdCR.SelForce;
END_REGION

REGION Network 14: **** 2.2 - Alarms - Alarms Generation **** STOP is selected in control room
   #AD_SelStop := #HMICmdCR.SelStop;
END_REGION

REGION Network 15: **** 2.2 - Alarms - Alarms Generation **** RELIEF is selected in control room
   #AD_SelRelief := #HMICmdCR.SelRelief;
END_REGION

REGION Network 16: **** 4.4 MachineStatus - Calculated **** DateTime PLC
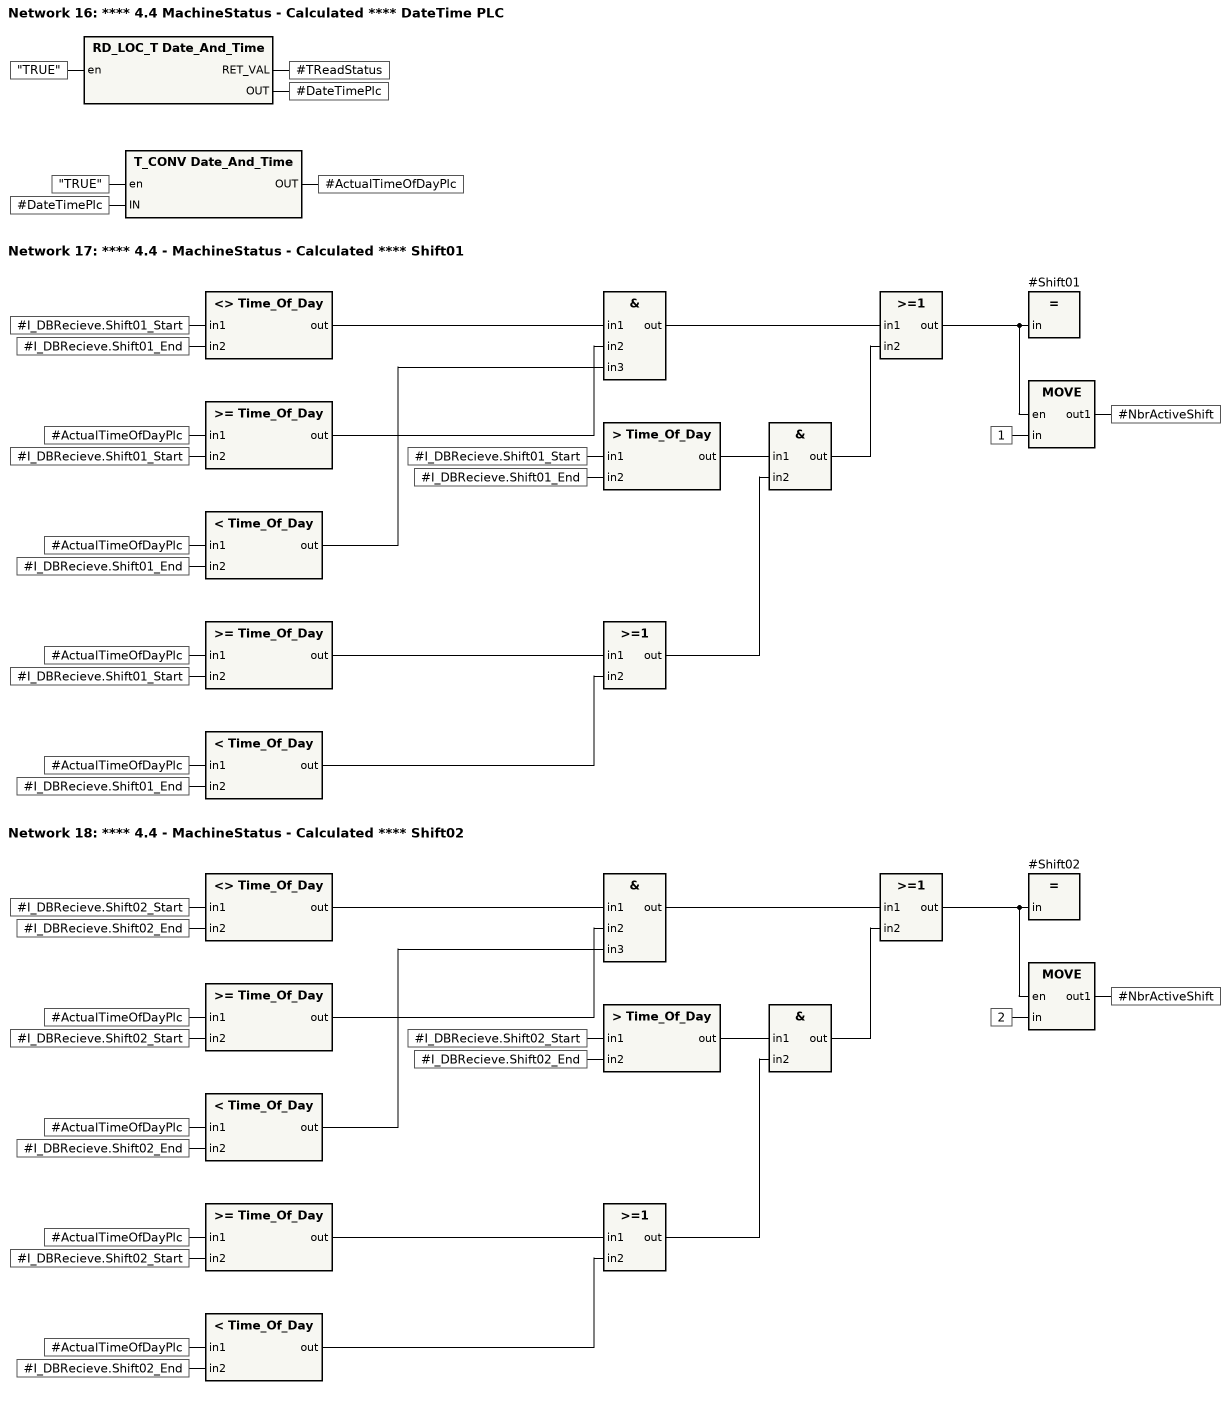
   IF "TRUE" THEN #TReadStatus := RD_LOC_T(OUT => #DateTimePlc); END_IF;
   IF "TRUE" THEN T_CONV(IN := #DateTimePlc, OUT => #ActualTimeOfDayPlc); END_IF;
END_REGION

REGION Network 17: **** 4.4 - MachineStatus - Calculated **** Shift01
   #Shift01 := ((#I_DBRecieve.Shift01_Start <> #I_DBRecieve.Shift01_End) AND (#ActualTimeOfDayPlc >= #I_DBRecieve.Shift01_Start) AND (#ActualTimeOfDayPlc < #I_DBRecieve.Shift01_End)) OR ((#I_DBRecieve.Shift01_Start > #I_DBRecieve.Shift01_End) AND ((#ActualTimeOfDayPlc >= #I_DBRecieve.Shift01_Start) OR (#ActualTimeOfDayPlc < #I_DBRecieve.Shift01_End)));
   IF #Shift01 THEN #NbrActiveShift := 1; END_IF;
END_REGION

REGION Network 18: **** 4.4 - MachineStatus - Calculated **** Shift02
   #Shift02 := ((#I_DBRecieve.Shift02_Start <> #I_DBRecieve.Shift02_End) AND (#ActualTimeOfDayPlc >= #I_DBRecieve.Shift02_Start) AND (#ActualTimeOfDayPlc < #I_DBRecieve.Shift02_End)) OR ((#I_DBRecieve.Shift02_Start > #I_DBRecieve.Shift02_End) AND ((#ActualTimeOfDayPlc >= #I_DBRecieve.Shift02_Start) OR (#ActualTimeOfDayPlc < #I_DBRecieve.Shift02_End)));
   IF #Shift02 THEN #NbrActiveShift := 2; END_IF;
END_REGION

REGION Network 19: **** 4.4 - MachineStatus - Calculated **** Shift03
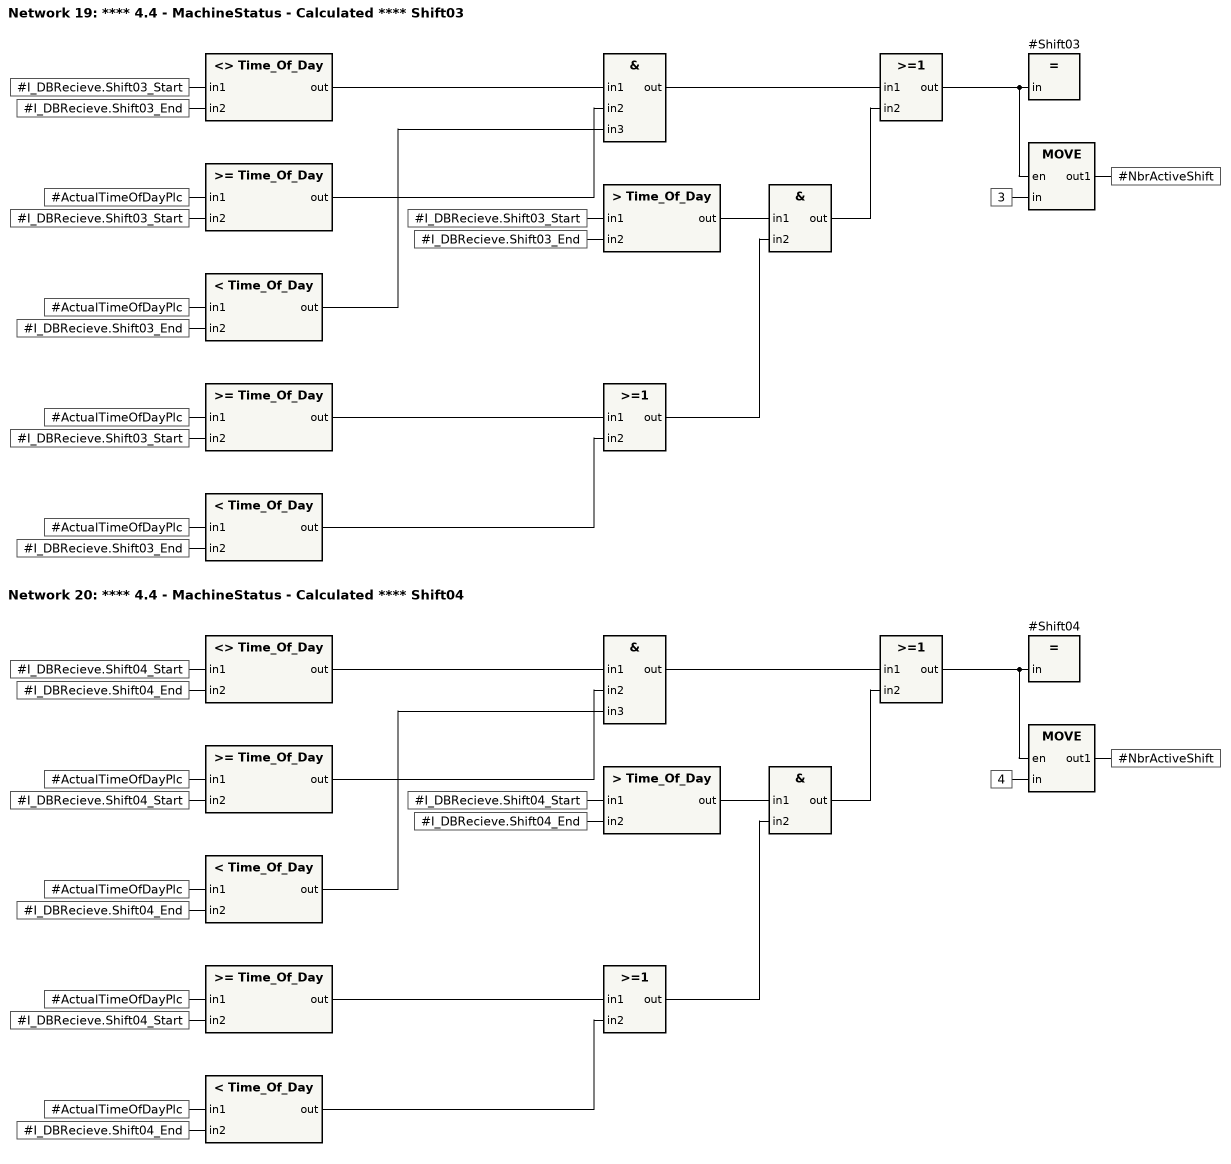
   #Shift03 := ((#I_DBRecieve.Shift03_Start <> #I_DBRecieve.Shift03_End) AND (#ActualTimeOfDayPlc >= #I_DBRecieve.Shift03_Start) AND (#ActualTimeOfDayPlc < #I_DBRecieve.Shift03_End)) OR ((#I_DBRecieve.Shift03_Start > #I_DBRecieve.Shift03_End) AND ((#ActualTimeOfDayPlc >= #I_DBRecieve.Shift03_Start) OR (#ActualTimeOfDayPlc < #I_DBRecieve.Shift03_End)));
   IF #Shift03 THEN #NbrActiveShift := 3; END_IF;
END_REGION

REGION Network 20: **** 4.4 - MachineStatus - Calculated **** Shift04
   #Shift04 := ((#I_DBRecieve.Shift04_Start <> #I_DBRecieve.Shift04_End) AND (#ActualTimeOfDayPlc >= #I_DBRecieve.Shift04_Start) AND (#ActualTimeOfDayPlc < #I_DBRecieve.Shift04_End)) OR ((#I_DBRecieve.Shift04_Start > #I_DBRecieve.Shift04_End) AND ((#ActualTimeOfDayPlc >= #I_DBRecieve.Shift04_Start) OR (#ActualTimeOfDayPlc < #I_DBRecieve.Shift04_End)));
   IF #Shift04 THEN #NbrActiveShift := 4; END_IF;
END_REGION

REGION Network 21: **** 4.4 - MachineStatus - Calculated **** Shift05
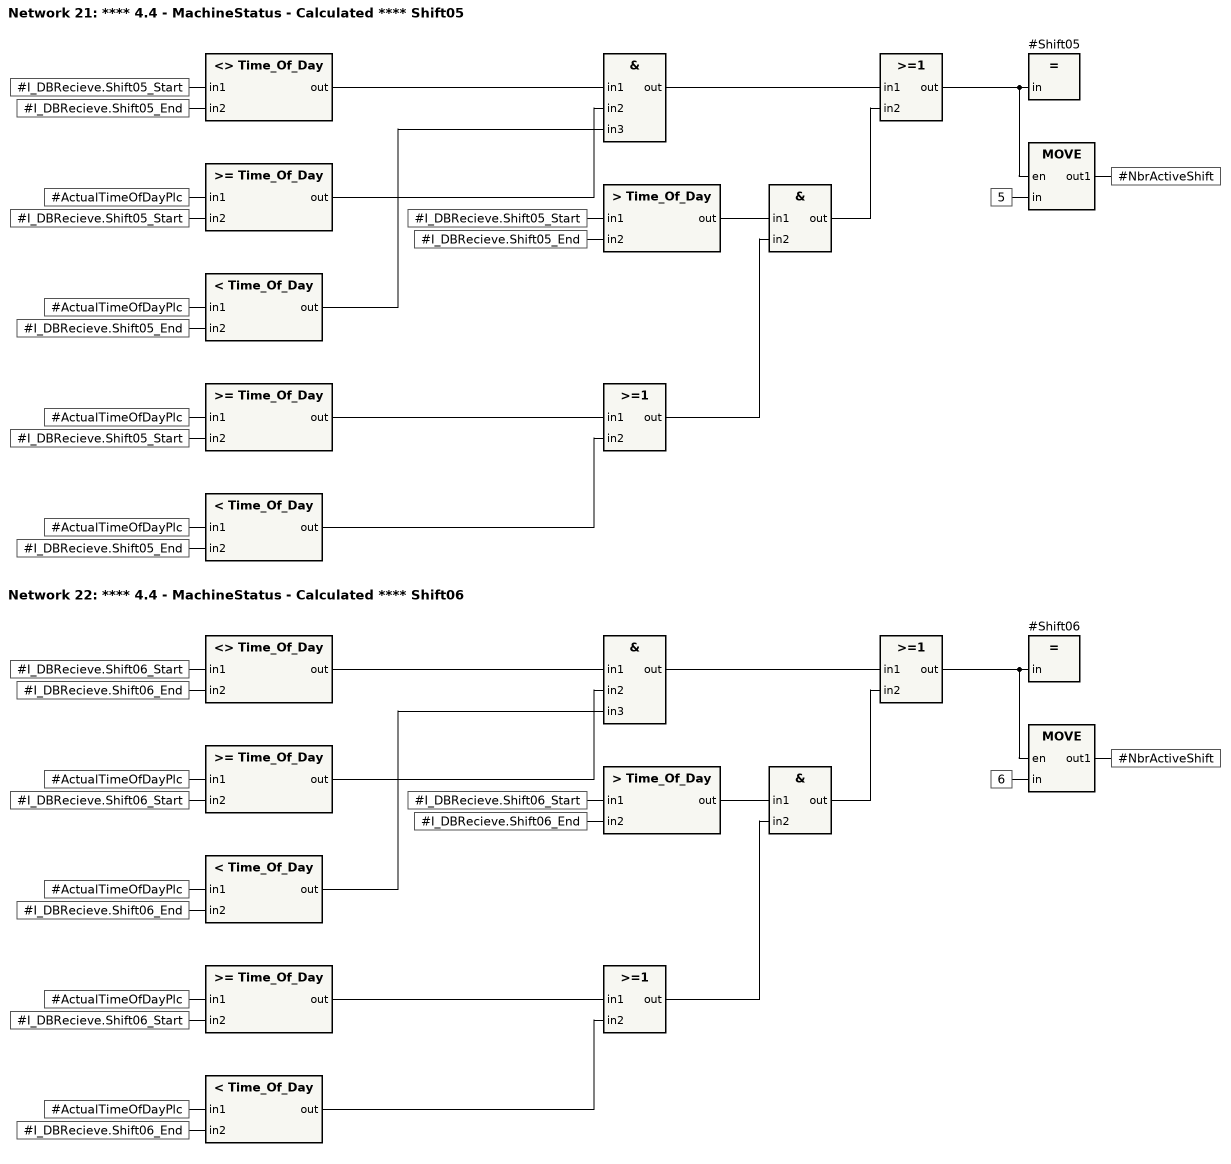
   #Shift05 := ((#I_DBRecieve.Shift05_Start <> #I_DBRecieve.Shift05_End) AND (#ActualTimeOfDayPlc >= #I_DBRecieve.Shift05_Start) AND (#ActualTimeOfDayPlc < #I_DBRecieve.Shift05_End)) OR ((#I_DBRecieve.Shift05_Start > #I_DBRecieve.Shift05_End) AND ((#ActualTimeOfDayPlc >= #I_DBRecieve.Shift05_Start) OR (#ActualTimeOfDayPlc < #I_DBRecieve.Shift05_End)));
   IF #Shift05 THEN #NbrActiveShift := 5; END_IF;
END_REGION

REGION Network 22: **** 4.4 - MachineStatus - Calculated **** Shift06
   #Shift06 := ((#I_DBRecieve.Shift06_Start <> #I_DBRecieve.Shift06_End) AND (#ActualTimeOfDayPlc >= #I_DBRecieve.Shift06_Start) AND (#ActualTimeOfDayPlc < #I_DBRecieve.Shift06_End)) OR ((#I_DBRecieve.Shift06_Start > #I_DBRecieve.Shift06_End) AND ((#ActualTimeOfDayPlc >= #I_DBRecieve.Shift06_Start) OR (#ActualTimeOfDayPlc < #I_DBRecieve.Shift06_End)));
   IF #Shift06 THEN #NbrActiveShift := 6; END_IF;
END_REGION

REGION Network 23: **** 4.4 - MachineStatus - Calculated **** Break01
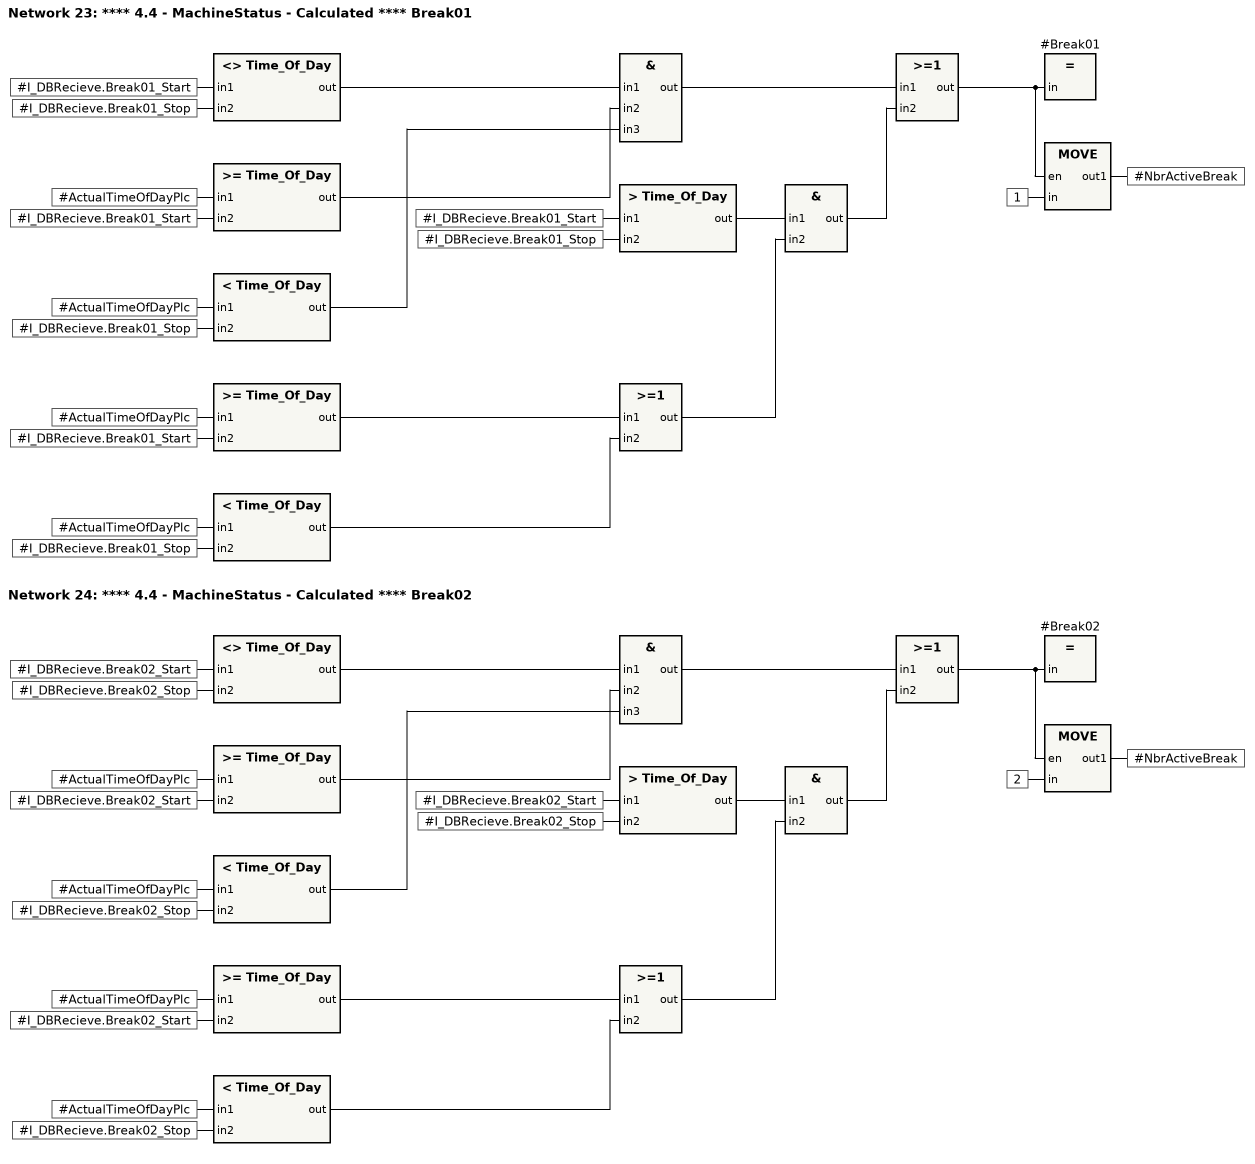
   #Break01 := ((#I_DBRecieve.Break01_Start <> #I_DBRecieve.Break01_Stop) AND (#ActualTimeOfDayPlc >= #I_DBRecieve.Break01_Start) AND (#ActualTimeOfDayPlc < #I_DBRecieve.Break01_Stop)) OR ((#I_DBRecieve.Break01_Start > #I_DBRecieve.Break01_Stop) AND ((#ActualTimeOfDayPlc >= #I_DBRecieve.Break01_Start) OR (#ActualTimeOfDayPlc < #I_DBRecieve.Break01_Stop)));
   IF #Break01 THEN #NbrActiveBreak := 1; END_IF;
END_REGION

REGION Network 24: **** 4.4 - MachineStatus - Calculated **** Break02
   #Break02 := ((#I_DBRecieve.Break02_Start <> #I_DBRecieve.Break02_Stop) AND (#ActualTimeOfDayPlc >= #I_DBRecieve.Break02_Start) AND (#ActualTimeOfDayPlc < #I_DBRecieve.Break02_Stop)) OR ((#I_DBRecieve.Break02_Start > #I_DBRecieve.Break02_Stop) AND ((#ActualTimeOfDayPlc >= #I_DBRecieve.Break02_Start) OR (#ActualTimeOfDayPlc < #I_DBRecieve.Break02_Stop)));
   IF #Break02 THEN #NbrActiveBreak := 2; END_IF;
END_REGION

REGION Network 25: **** 4.4 - MachineStatus - Calculated **** Break03
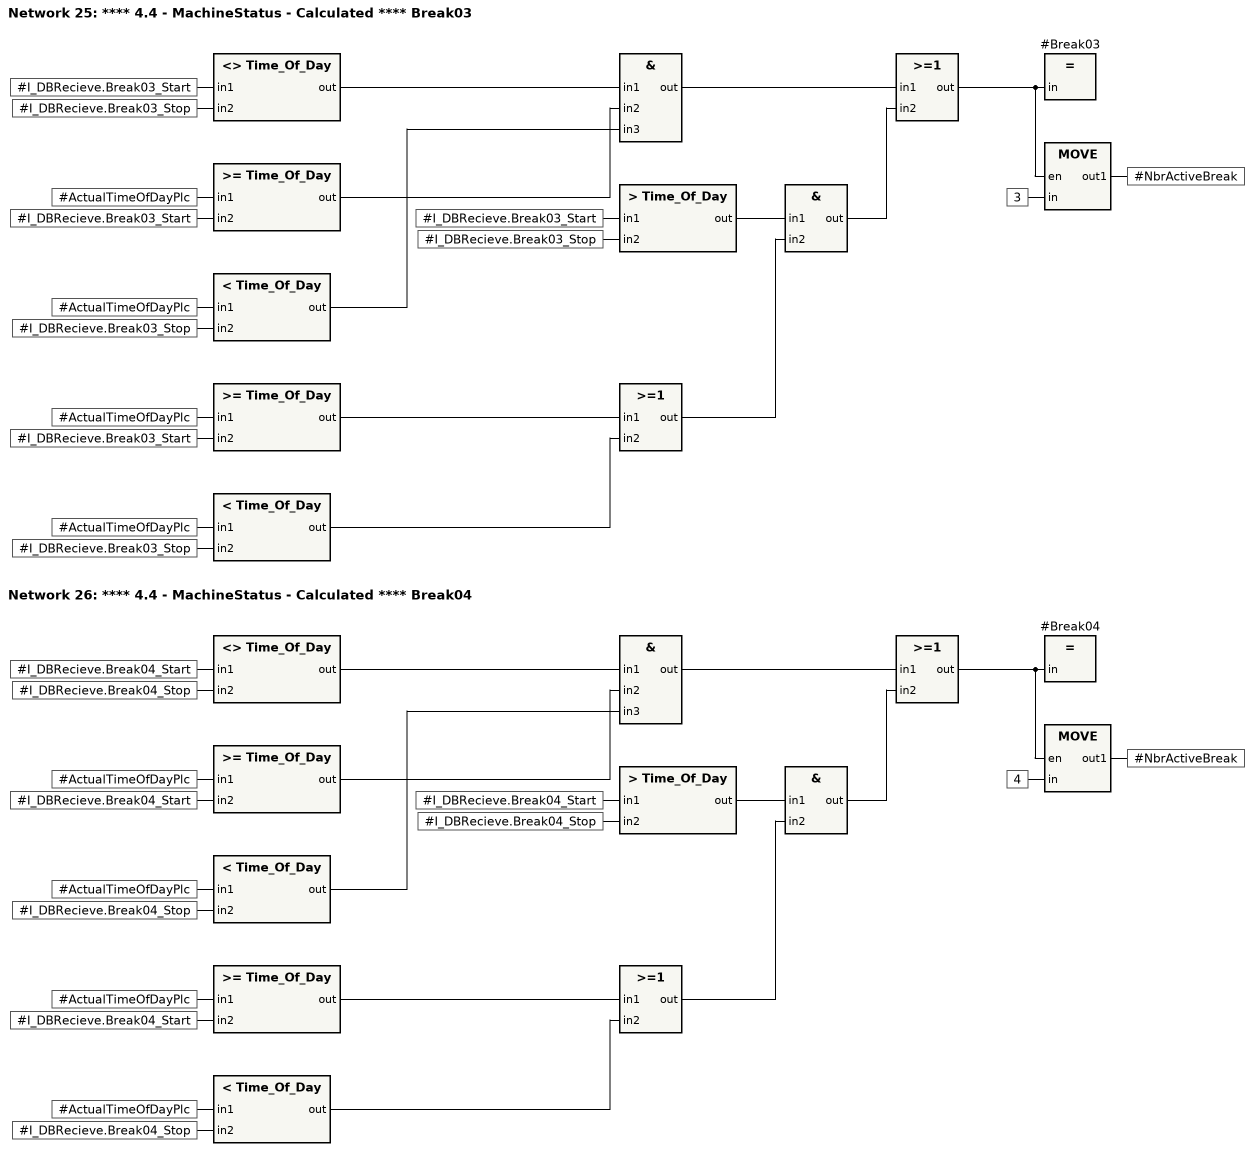
   #Break03 := ((#I_DBRecieve.Break03_Start <> #I_DBRecieve.Break03_Stop) AND (#ActualTimeOfDayPlc >= #I_DBRecieve.Break03_Start) AND (#ActualTimeOfDayPlc < #I_DBRecieve.Break03_Stop)) OR ((#I_DBRecieve.Break03_Start > #I_DBRecieve.Break03_Stop) AND ((#ActualTimeOfDayPlc >= #I_DBRecieve.Break03_Start) OR (#ActualTimeOfDayPlc < #I_DBRecieve.Break03_Stop)));
   IF #Break03 THEN #NbrActiveBreak := 3; END_IF;
END_REGION

REGION Network 26: **** 4.4 - MachineStatus - Calculated **** Break04
   #Break04 := ((#I_DBRecieve.Break04_Start <> #I_DBRecieve.Break04_Stop) AND (#ActualTimeOfDayPlc >= #I_DBRecieve.Break04_Start) AND (#ActualTimeOfDayPlc < #I_DBRecieve.Break04_Stop)) OR ((#I_DBRecieve.Break04_Start > #I_DBRecieve.Break04_Stop) AND ((#ActualTimeOfDayPlc >= #I_DBRecieve.Break04_Start) OR (#ActualTimeOfDayPlc < #I_DBRecieve.Break04_Stop)));
   IF #Break04 THEN #NbrActiveBreak := 4; END_IF;
END_REGION

REGION Network 27: **** 4.4 - MachineStatus - Calculated **** Break05
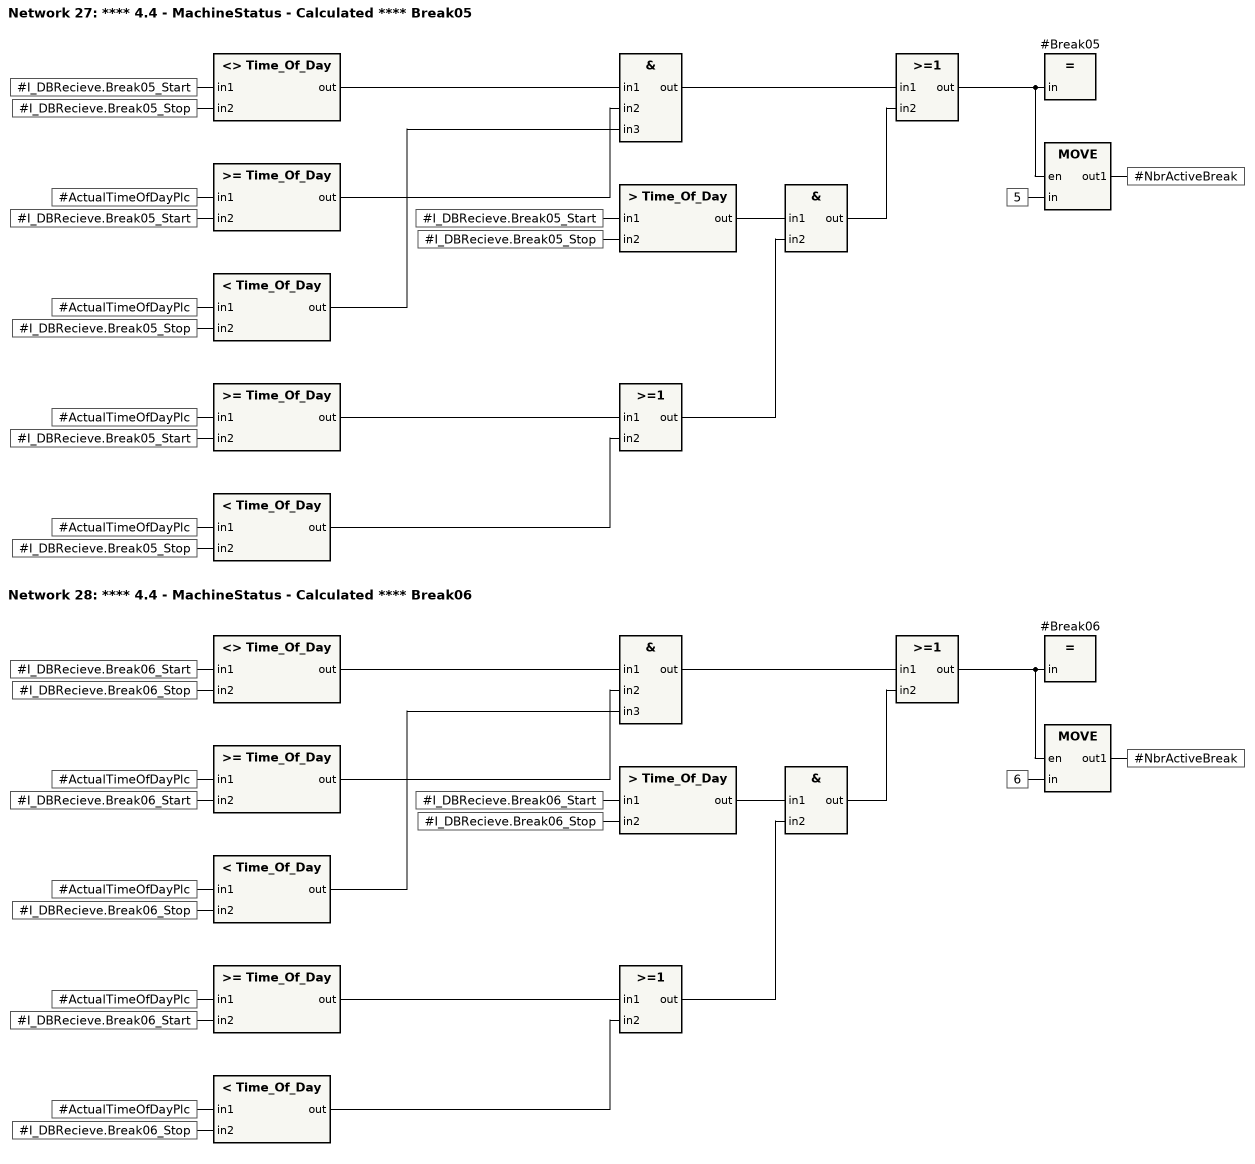
   #Break05 := ((#I_DBRecieve.Break05_Start <> #I_DBRecieve.Break05_Stop) AND (#ActualTimeOfDayPlc >= #I_DBRecieve.Break05_Start) AND (#ActualTimeOfDayPlc < #I_DBRecieve.Break05_Stop)) OR ((#I_DBRecieve.Break05_Start > #I_DBRecieve.Break05_Stop) AND ((#ActualTimeOfDayPlc >= #I_DBRecieve.Break05_Start) OR (#ActualTimeOfDayPlc < #I_DBRecieve.Break05_Stop)));
   IF #Break05 THEN #NbrActiveBreak := 5; END_IF;
END_REGION

REGION Network 28: **** 4.4 - MachineStatus - Calculated **** Break06
   #Break06 := ((#I_DBRecieve.Break06_Start <> #I_DBRecieve.Break06_Stop) AND (#ActualTimeOfDayPlc >= #I_DBRecieve.Break06_Start) AND (#ActualTimeOfDayPlc < #I_DBRecieve.Break06_Stop)) OR ((#I_DBRecieve.Break06_Start > #I_DBRecieve.Break06_Stop) AND ((#ActualTimeOfDayPlc >= #I_DBRecieve.Break06_Start) OR (#ActualTimeOfDayPlc < #I_DBRecieve.Break06_Stop)));
   IF #Break06 THEN #NbrActiveBreak := 6; END_IF;
END_REGION

REGION Network 29: **** 4.4 - MachineStatus - Calculated **** Morning Shift Rotation01
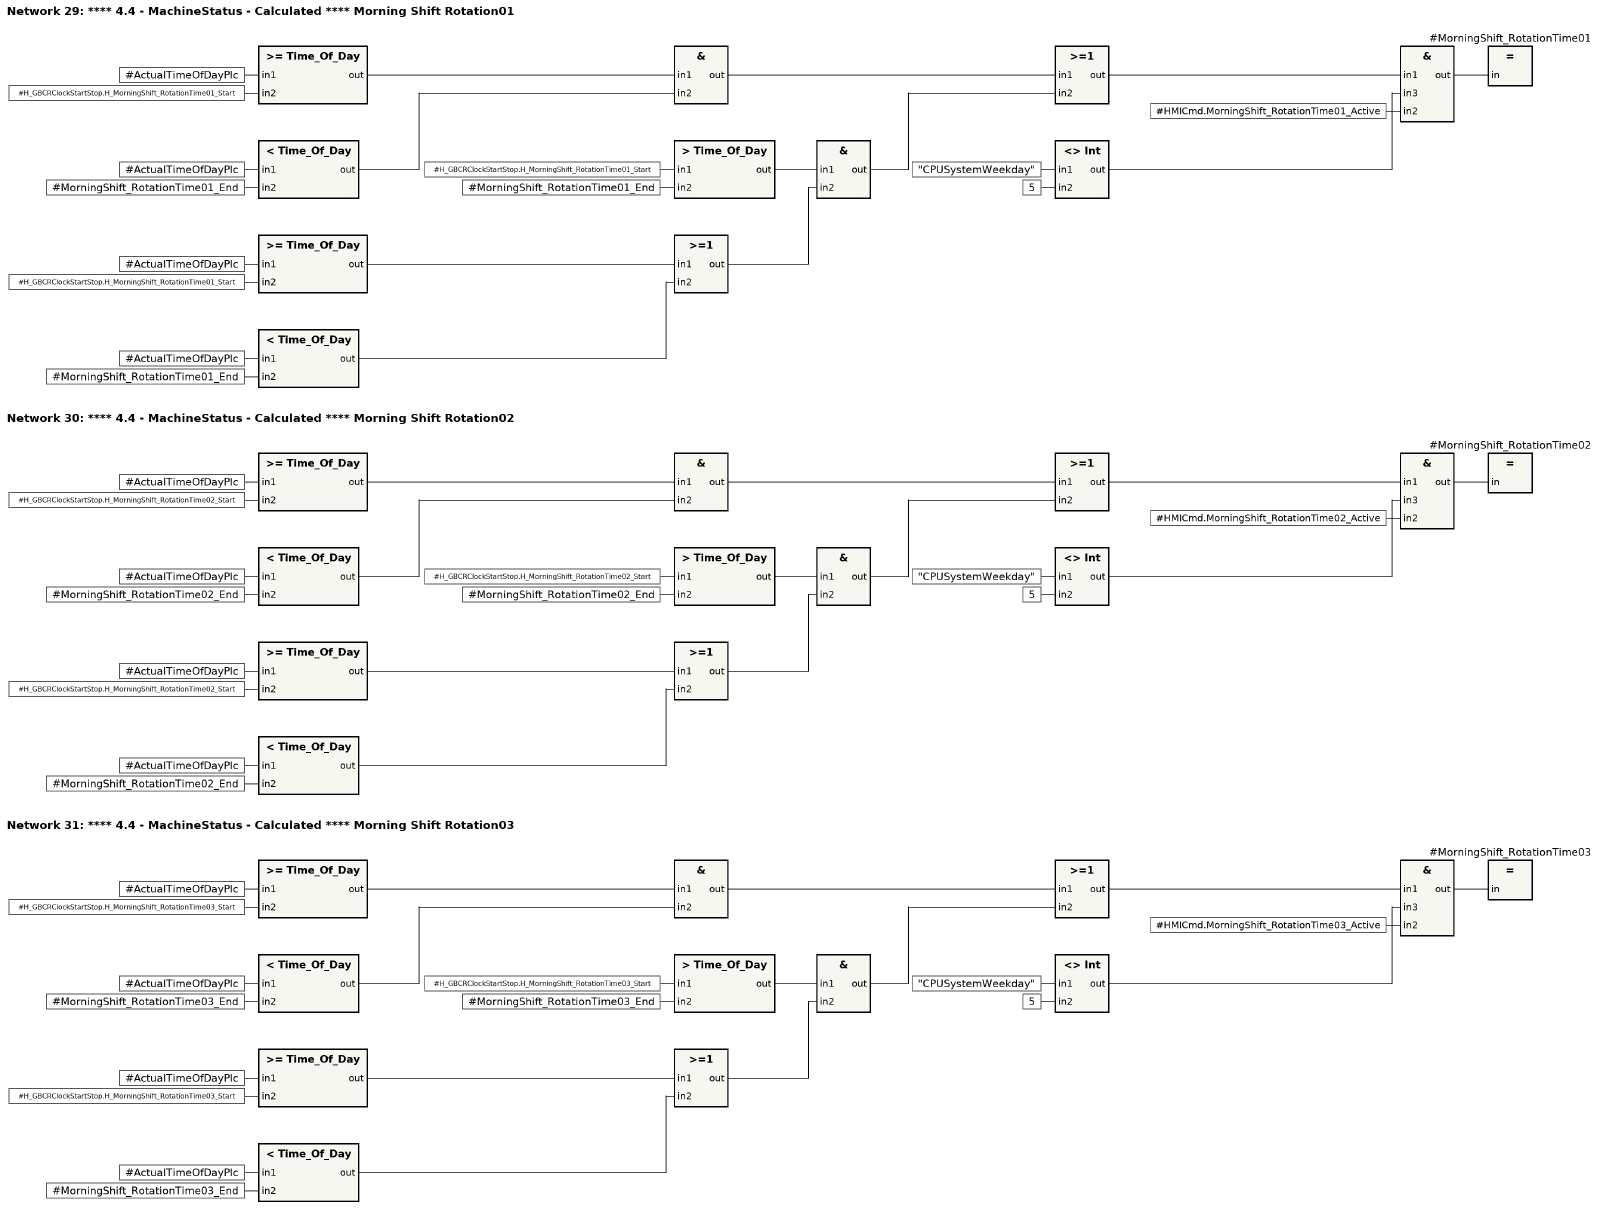
   #MorningShift_RotationTime01 := (((#ActualTimeOfDayPlc >= #H_GBCRClockStartStop.H_MorningShift_RotationTime01_Start) AND (#ActualTimeOfDayPlc < #MorningShift_RotationTime01_End)) OR ((#H_GBCRClockStartStop.H_MorningShift_RotationTime01_Start > #MorningShift_RotationTime01_End) AND ((#ActualTimeOfDayPlc >= #H_GBCRClockStartStop.H_MorningShift_RotationTime01_Start) OR (#ActualTimeOfDayPlc < #MorningShift_RotationTime01_End)))) AND ("CPUSystemWeekday" <> 5) AND #HMICmd.MorningShift_RotationTime01_Active;
END_REGION

REGION Network 30: **** 4.4 - MachineStatus - Calculated **** Morning Shift Rotation02
   #MorningShift_RotationTime02 := (((#ActualTimeOfDayPlc >= #H_GBCRClockStartStop.H_MorningShift_RotationTime02_Start) AND (#ActualTimeOfDayPlc < #MorningShift_RotationTime02_End)) OR ((#H_GBCRClockStartStop.H_MorningShift_RotationTime02_Start > #MorningShift_RotationTime02_End) AND ((#ActualTimeOfDayPlc >= #H_GBCRClockStartStop.H_MorningShift_RotationTime02_Start) OR (#ActualTimeOfDayPlc < #MorningShift_RotationTime02_End)))) AND ("CPUSystemWeekday" <> 5) AND #HMICmd.MorningShift_RotationTime02_Active;
END_REGION

REGION Network 31: **** 4.4 - MachineStatus - Calculated **** Morning Shift Rotation03
   #MorningShift_RotationTime03 := (((#ActualTimeOfDayPlc >= #H_GBCRClockStartStop.H_MorningShift_RotationTime03_Start) AND (#ActualTimeOfDayPlc < #MorningShift_RotationTime03_End)) OR ((#H_GBCRClockStartStop.H_MorningShift_RotationTime03_Start > #MorningShift_RotationTime03_End) AND ((#ActualTimeOfDayPlc >= #H_GBCRClockStartStop.H_MorningShift_RotationTime03_Start) OR (#ActualTimeOfDayPlc < #MorningShift_RotationTime03_End)))) AND ("CPUSystemWeekday" <> 5) AND #HMICmd.MorningShift_RotationTime03_Active;
END_REGION

REGION Network 32: **** 4.4 - MachineStatus - Calculated **** Morning Shift Rotation04
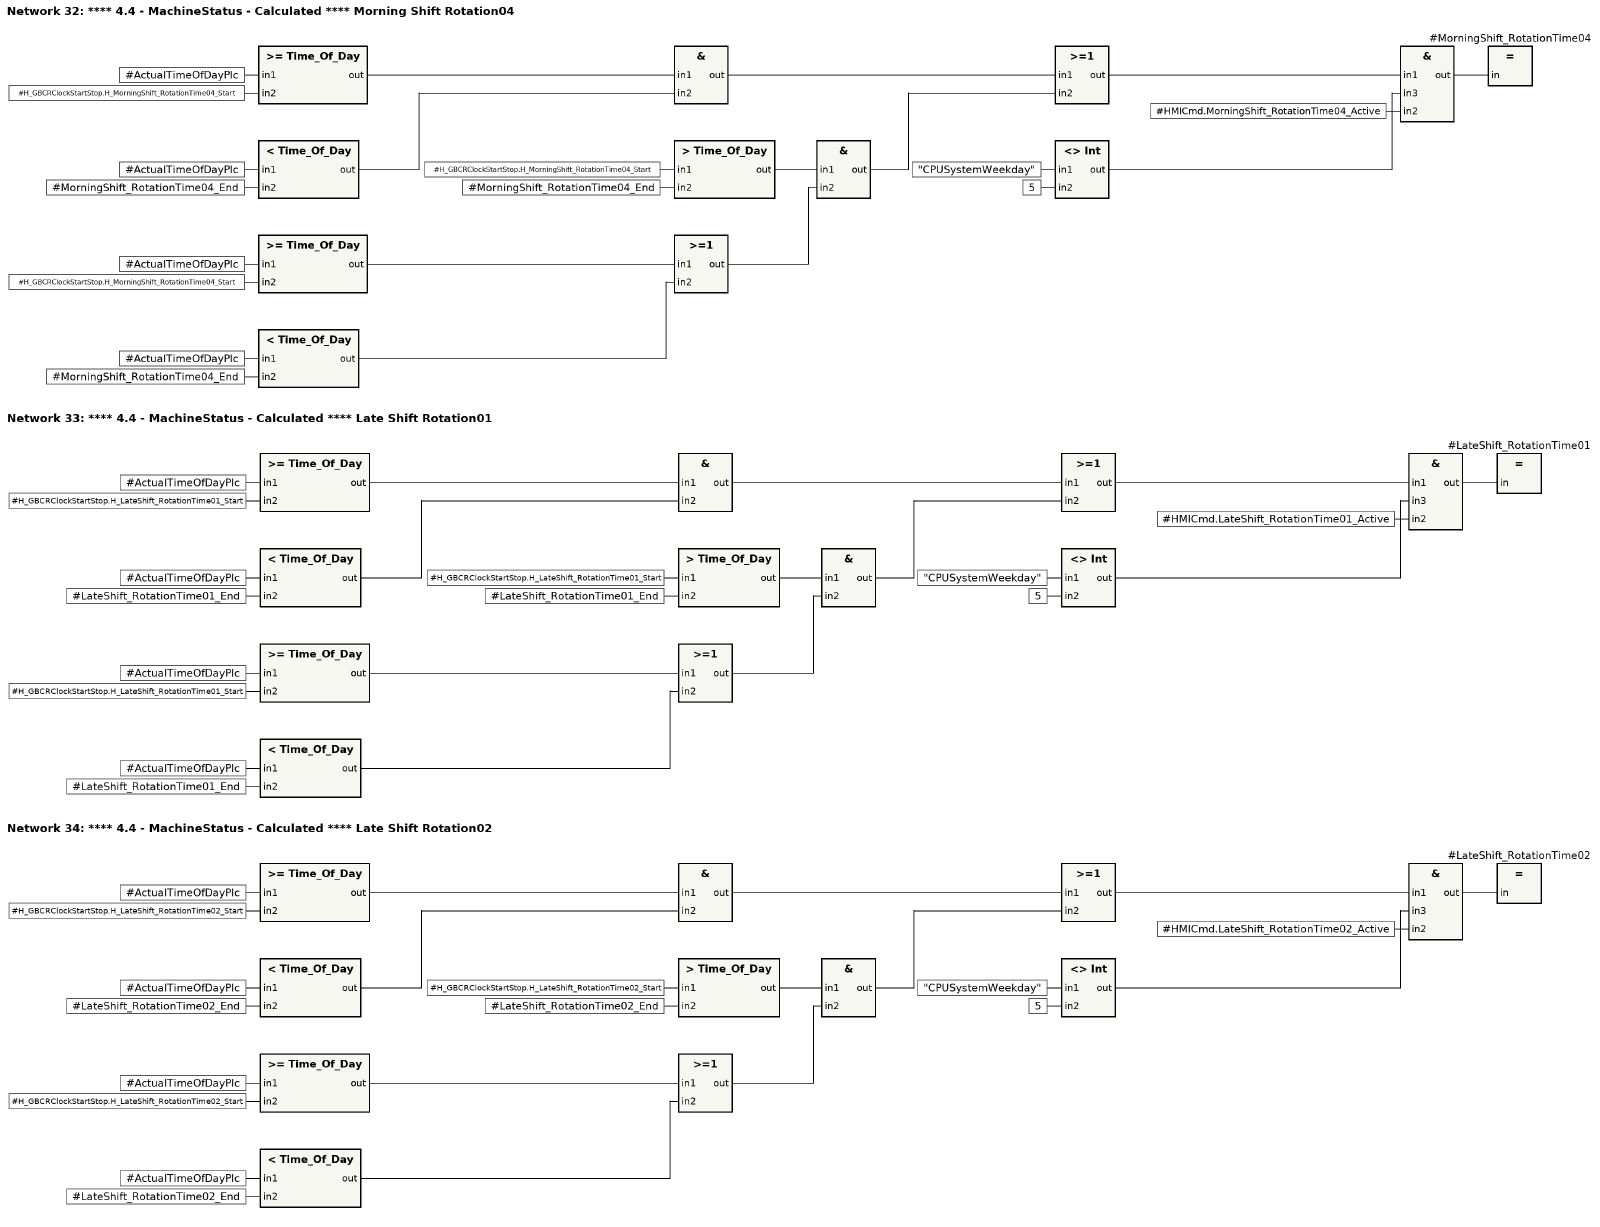
   #MorningShift_RotationTime04 := (((#ActualTimeOfDayPlc >= #H_GBCRClockStartStop.H_MorningShift_RotationTime04_Start) AND (#ActualTimeOfDayPlc < #MorningShift_RotationTime04_End)) OR ((#H_GBCRClockStartStop.H_MorningShift_RotationTime04_Start > #MorningShift_RotationTime04_End) AND ((#ActualTimeOfDayPlc >= #H_GBCRClockStartStop.H_MorningShift_RotationTime04_Start) OR (#ActualTimeOfDayPlc < #MorningShift_RotationTime04_End)))) AND ("CPUSystemWeekday" <> 5) AND #HMICmd.MorningShift_RotationTime04_Active;
END_REGION

REGION Network 33: **** 4.4 - MachineStatus - Calculated **** Late Shift Rotation01
   #LateShift_RotationTime01 := (((#ActualTimeOfDayPlc >= #H_GBCRClockStartStop.H_LateShift_RotationTime01_Start) AND (#ActualTimeOfDayPlc < #LateShift_RotationTime01_End)) OR ((#H_GBCRClockStartStop.H_LateShift_RotationTime01_Start > #LateShift_RotationTime01_End) AND ((#ActualTimeOfDayPlc >= #H_GBCRClockStartStop.H_LateShift_RotationTime01_Start) OR (#ActualTimeOfDayPlc < #LateShift_RotationTime01_End)))) AND ("CPUSystemWeekday" <> 5) AND #HMICmd.LateShift_RotationTime01_Active;
END_REGION

REGION Network 34: **** 4.4 - MachineStatus - Calculated **** Late Shift Rotation02
   #LateShift_RotationTime02 := (((#ActualTimeOfDayPlc >= #H_GBCRClockStartStop.H_LateShift_RotationTime02_Start) AND (#ActualTimeOfDayPlc < #LateShift_RotationTime02_End)) OR ((#H_GBCRClockStartStop.H_LateShift_RotationTime02_Start > #LateShift_RotationTime02_End) AND ((#ActualTimeOfDayPlc >= #H_GBCRClockStartStop.H_LateShift_RotationTime02_Start) OR (#ActualTimeOfDayPlc < #LateShift_RotationTime02_End)))) AND ("CPUSystemWeekday" <> 5) AND #HMICmd.LateShift_RotationTime02_Active;
END_REGION

REGION Network 35: **** 4.4 - MachineStatus - Calculated **** Late Shift Rotation03
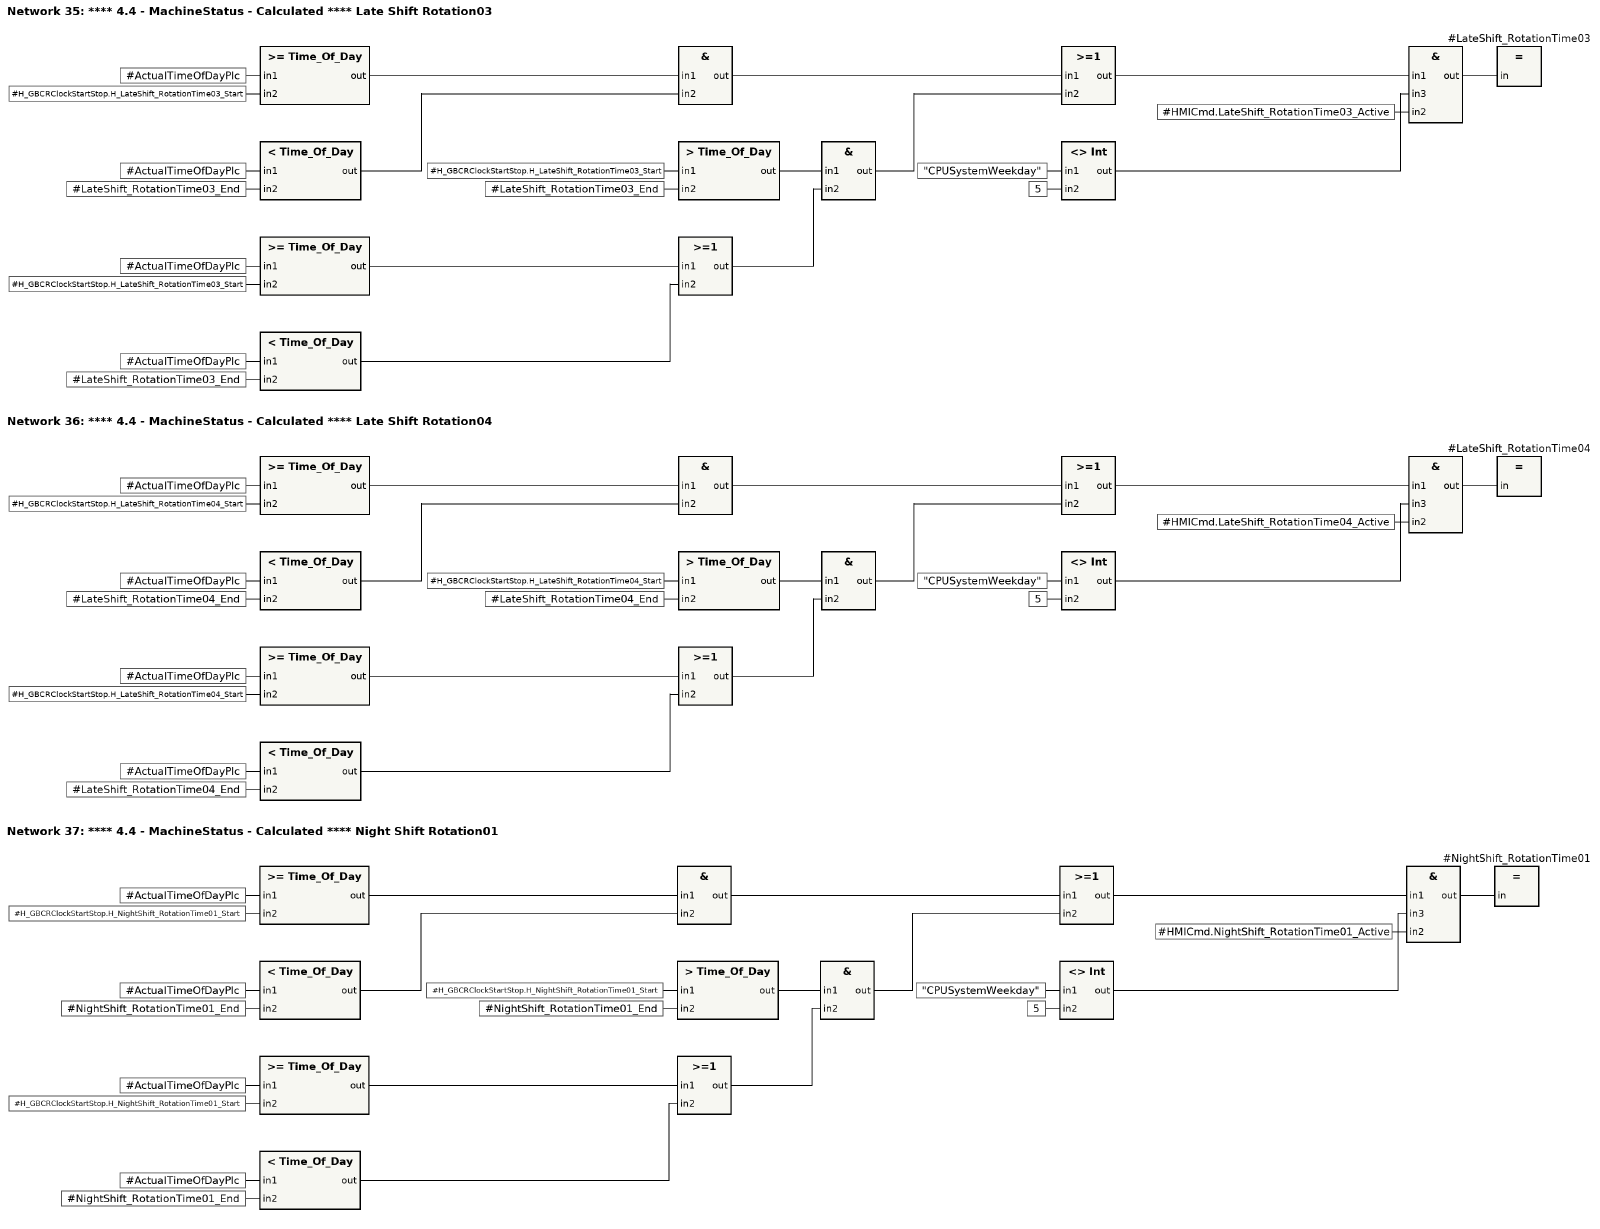
   #LateShift_RotationTime03 := (((#ActualTimeOfDayPlc >= #H_GBCRClockStartStop.H_LateShift_RotationTime03_Start) AND (#ActualTimeOfDayPlc < #LateShift_RotationTime03_End)) OR ((#H_GBCRClockStartStop.H_LateShift_RotationTime03_Start > #LateShift_RotationTime03_End) AND ((#ActualTimeOfDayPlc >= #H_GBCRClockStartStop.H_LateShift_RotationTime03_Start) OR (#ActualTimeOfDayPlc < #LateShift_RotationTime03_End)))) AND ("CPUSystemWeekday" <> 5) AND #HMICmd.LateShift_RotationTime03_Active;
END_REGION

REGION Network 36: **** 4.4 - MachineStatus - Calculated **** Late Shift Rotation04
   #LateShift_RotationTime04 := (((#ActualTimeOfDayPlc >= #H_GBCRClockStartStop.H_LateShift_RotationTime04_Start) AND (#ActualTimeOfDayPlc < #LateShift_RotationTime04_End)) OR ((#H_GBCRClockStartStop.H_LateShift_RotationTime04_Start > #LateShift_RotationTime04_End) AND ((#ActualTimeOfDayPlc >= #H_GBCRClockStartStop.H_LateShift_RotationTime04_Start) OR (#ActualTimeOfDayPlc < #LateShift_RotationTime04_End)))) AND ("CPUSystemWeekday" <> 5) AND #HMICmd.LateShift_RotationTime04_Active;
END_REGION

REGION Network 37: **** 4.4 - MachineStatus - Calculated **** Night Shift Rotation01
   #NightShift_RotationTime01 := (((#ActualTimeOfDayPlc >= #H_GBCRClockStartStop.H_NightShift_RotationTime01_Start) AND (#ActualTimeOfDayPlc < #NightShift_RotationTime01_End)) OR ((#H_GBCRClockStartStop.H_NightShift_RotationTime01_Start > #NightShift_RotationTime01_End) AND ((#ActualTimeOfDayPlc >= #H_GBCRClockStartStop.H_NightShift_RotationTime01_Start) OR (#ActualTimeOfDayPlc < #NightShift_RotationTime01_End)))) AND ("CPUSystemWeekday" <> 5) AND #HMICmd.NightShift_RotationTime01_Active;
END_REGION

REGION Network 38: **** 4.4 - MachineStatus - Calculated **** Night Shift Rotation02
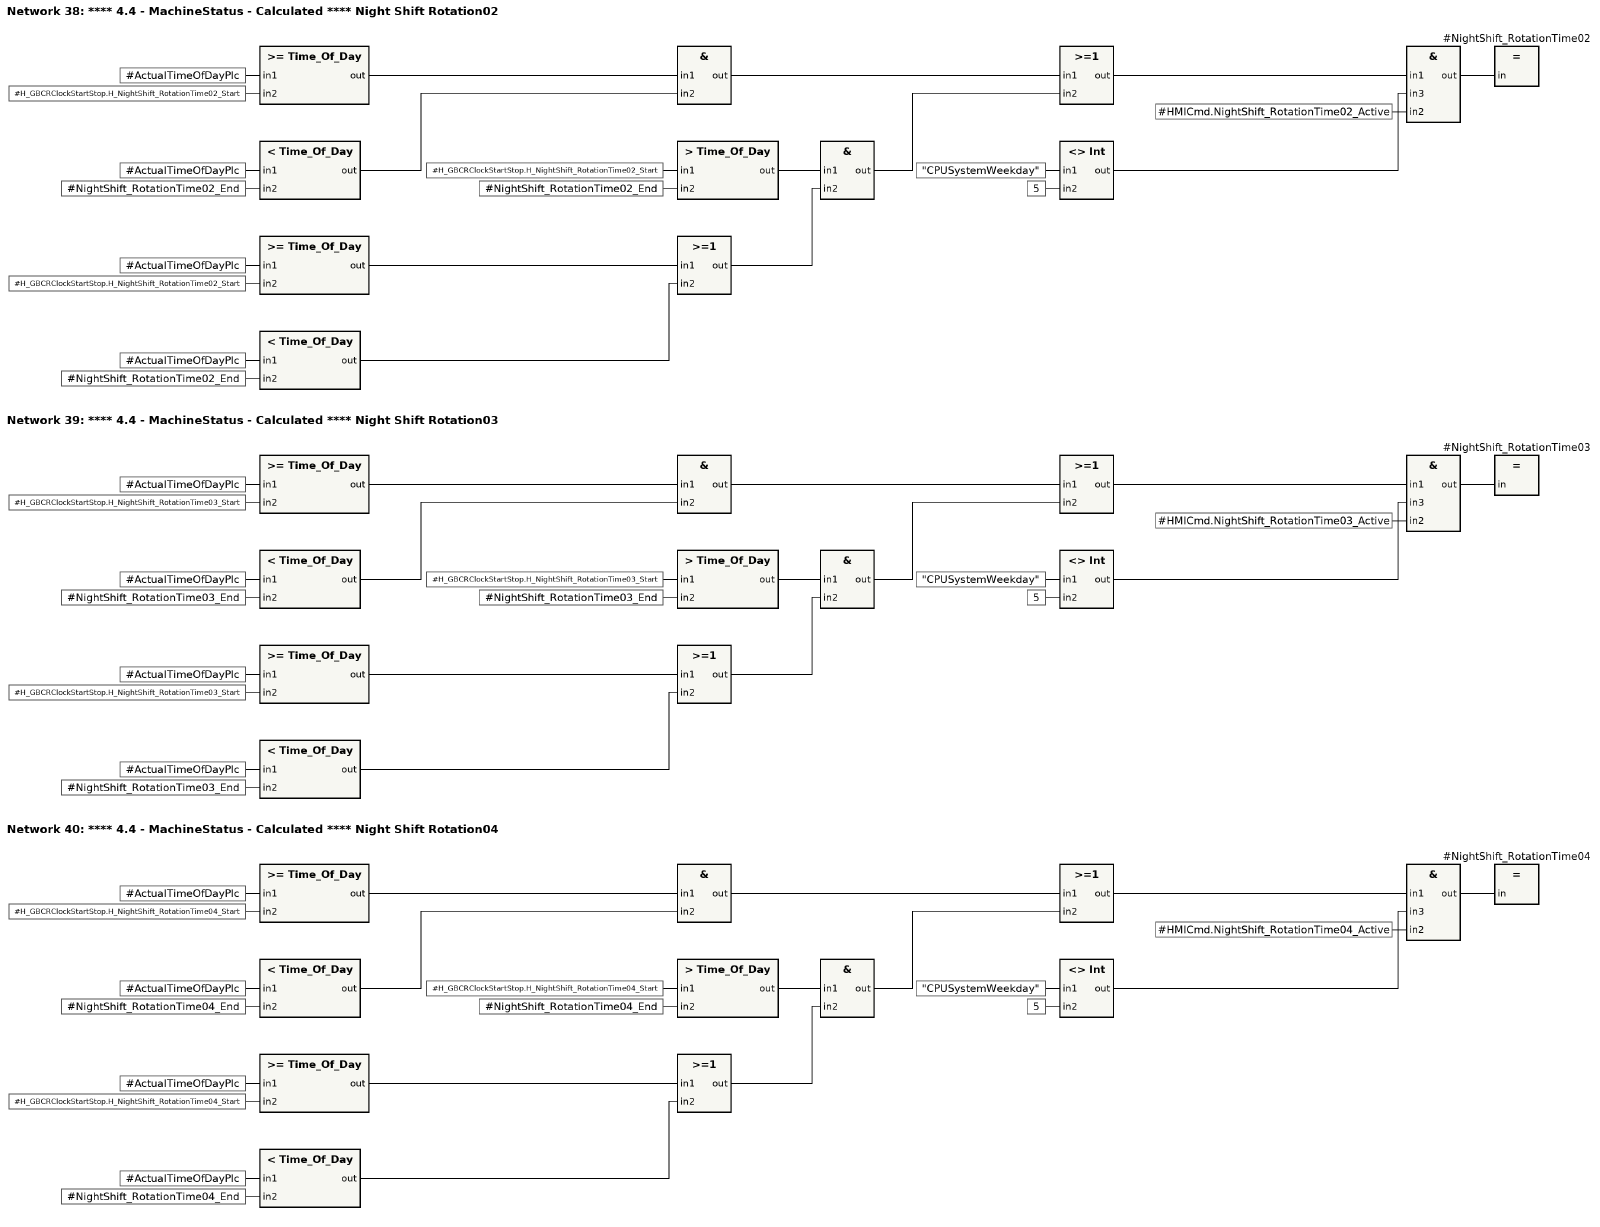
   #NightShift_RotationTime02 := (((#ActualTimeOfDayPlc >= #H_GBCRClockStartStop.H_NightShift_RotationTime02_Start) AND (#ActualTimeOfDayPlc < #NightShift_RotationTime02_End)) OR ((#H_GBCRClockStartStop.H_NightShift_RotationTime02_Start > #NightShift_RotationTime02_End) AND ((#ActualTimeOfDayPlc >= #H_GBCRClockStartStop.H_NightShift_RotationTime02_Start) OR (#ActualTimeOfDayPlc < #NightShift_RotationTime02_End)))) AND ("CPUSystemWeekday" <> 5) AND #HMICmd.NightShift_RotationTime02_Active;
END_REGION

REGION Network 39: **** 4.4 - MachineStatus - Calculated **** Night Shift Rotation03
   #NightShift_RotationTime03 := (((#ActualTimeOfDayPlc >= #H_GBCRClockStartStop.H_NightShift_RotationTime03_Start) AND (#ActualTimeOfDayPlc < #NightShift_RotationTime03_End)) OR ((#H_GBCRClockStartStop.H_NightShift_RotationTime03_Start > #NightShift_RotationTime03_End) AND ((#ActualTimeOfDayPlc >= #H_GBCRClockStartStop.H_NightShift_RotationTime03_Start) OR (#ActualTimeOfDayPlc < #NightShift_RotationTime03_End)))) AND ("CPUSystemWeekday" <> 5) AND #HMICmd.NightShift_RotationTime03_Active;
END_REGION

REGION Network 40: **** 4.4 - MachineStatus - Calculated **** Night Shift Rotation04
   #NightShift_RotationTime04 := (((#ActualTimeOfDayPlc >= #H_GBCRClockStartStop.H_NightShift_RotationTime04_Start) AND (#ActualTimeOfDayPlc < #NightShift_RotationTime04_End)) OR ((#H_GBCRClockStartStop.H_NightShift_RotationTime04_Start > #NightShift_RotationTime04_End) AND ((#ActualTimeOfDayPlc >= #H_GBCRClockStartStop.H_NightShift_RotationTime04_Start) OR (#ActualTimeOfDayPlc < #NightShift_RotationTime04_End)))) AND ("CPUSystemWeekday" <> 5) AND #HMICmd.NightShift_RotationTime04_Active;
END_REGION

REGION Network 41: **** 4.4 - MachineStatus - Calculated **** Morning Shift Rotation01 -> Day 5
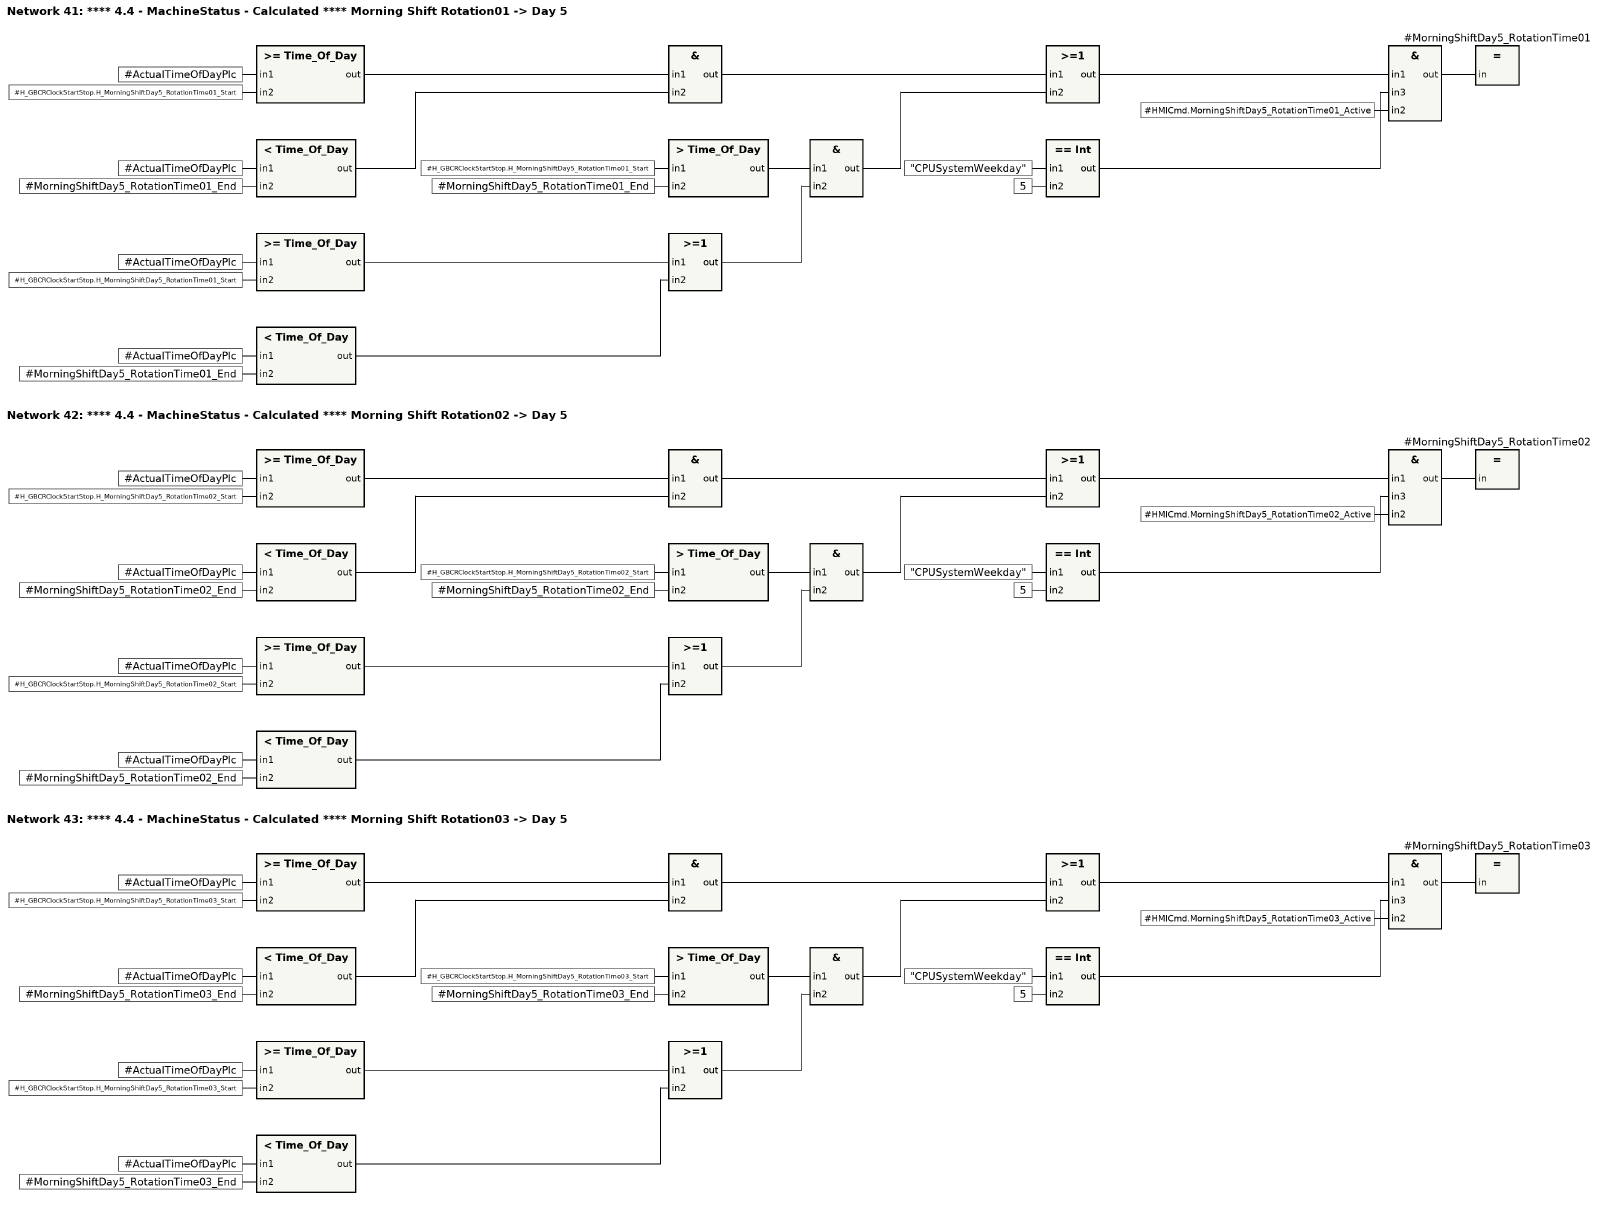
   #MorningShiftDay5_RotationTime01 := (((#ActualTimeOfDayPlc >= #H_GBCRClockStartStop.H_MorningShiftDay5_RotationTime01_Start) AND (#ActualTimeOfDayPlc < #MorningShiftDay5_RotationTime01_End)) OR ((#H_GBCRClockStartStop.H_MorningShiftDay5_RotationTime01_Start > #MorningShiftDay5_RotationTime01_End) AND ((#ActualTimeOfDayPlc >= #H_GBCRClockStartStop.H_MorningShiftDay5_RotationTime01_Start) OR (#ActualTimeOfDayPlc < #MorningShiftDay5_RotationTime01_End)))) AND ("CPUSystemWeekday" = 5) AND #HMICmd.MorningShiftDay5_RotationTime01_Active;
END_REGION

REGION Network 42: **** 4.4 - MachineStatus - Calculated **** Morning Shift Rotation02 -> Day 5
   #MorningShiftDay5_RotationTime02 := (((#ActualTimeOfDayPlc >= #H_GBCRClockStartStop.H_MorningShiftDay5_RotationTime02_Start) AND (#ActualTimeOfDayPlc < #MorningShiftDay5_RotationTime02_End)) OR ((#H_GBCRClockStartStop.H_MorningShiftDay5_RotationTime02_Start > #MorningShiftDay5_RotationTime02_End) AND ((#ActualTimeOfDayPlc >= #H_GBCRClockStartStop.H_MorningShiftDay5_RotationTime02_Start) OR (#ActualTimeOfDayPlc < #MorningShiftDay5_RotationTime02_End)))) AND ("CPUSystemWeekday" = 5) AND #HMICmd.MorningShiftDay5_RotationTime02_Active;
END_REGION

REGION Network 43: **** 4.4 - MachineStatus - Calculated **** Morning Shift Rotation03 -> Day 5
   #MorningShiftDay5_RotationTime03 := (((#ActualTimeOfDayPlc >= #H_GBCRClockStartStop.H_MorningShiftDay5_RotationTime03_Start) AND (#ActualTimeOfDayPlc < #MorningShiftDay5_RotationTime03_End)) OR ((#H_GBCRClockStartStop.H_MorningShiftDay5_RotationTime03_Start > #MorningShiftDay5_RotationTime03_End) AND ((#ActualTimeOfDayPlc >= #H_GBCRClockStartStop.H_MorningShiftDay5_RotationTime03_Start) OR (#ActualTimeOfDayPlc < #MorningShiftDay5_RotationTime03_End)))) AND ("CPUSystemWeekday" = 5) AND #HMICmd.MorningShiftDay5_RotationTime03_Active;
END_REGION

REGION Network 44: **** 4.4 - MachineStatus - Calculated **** Morning Shift Rotation04 -> Day 5
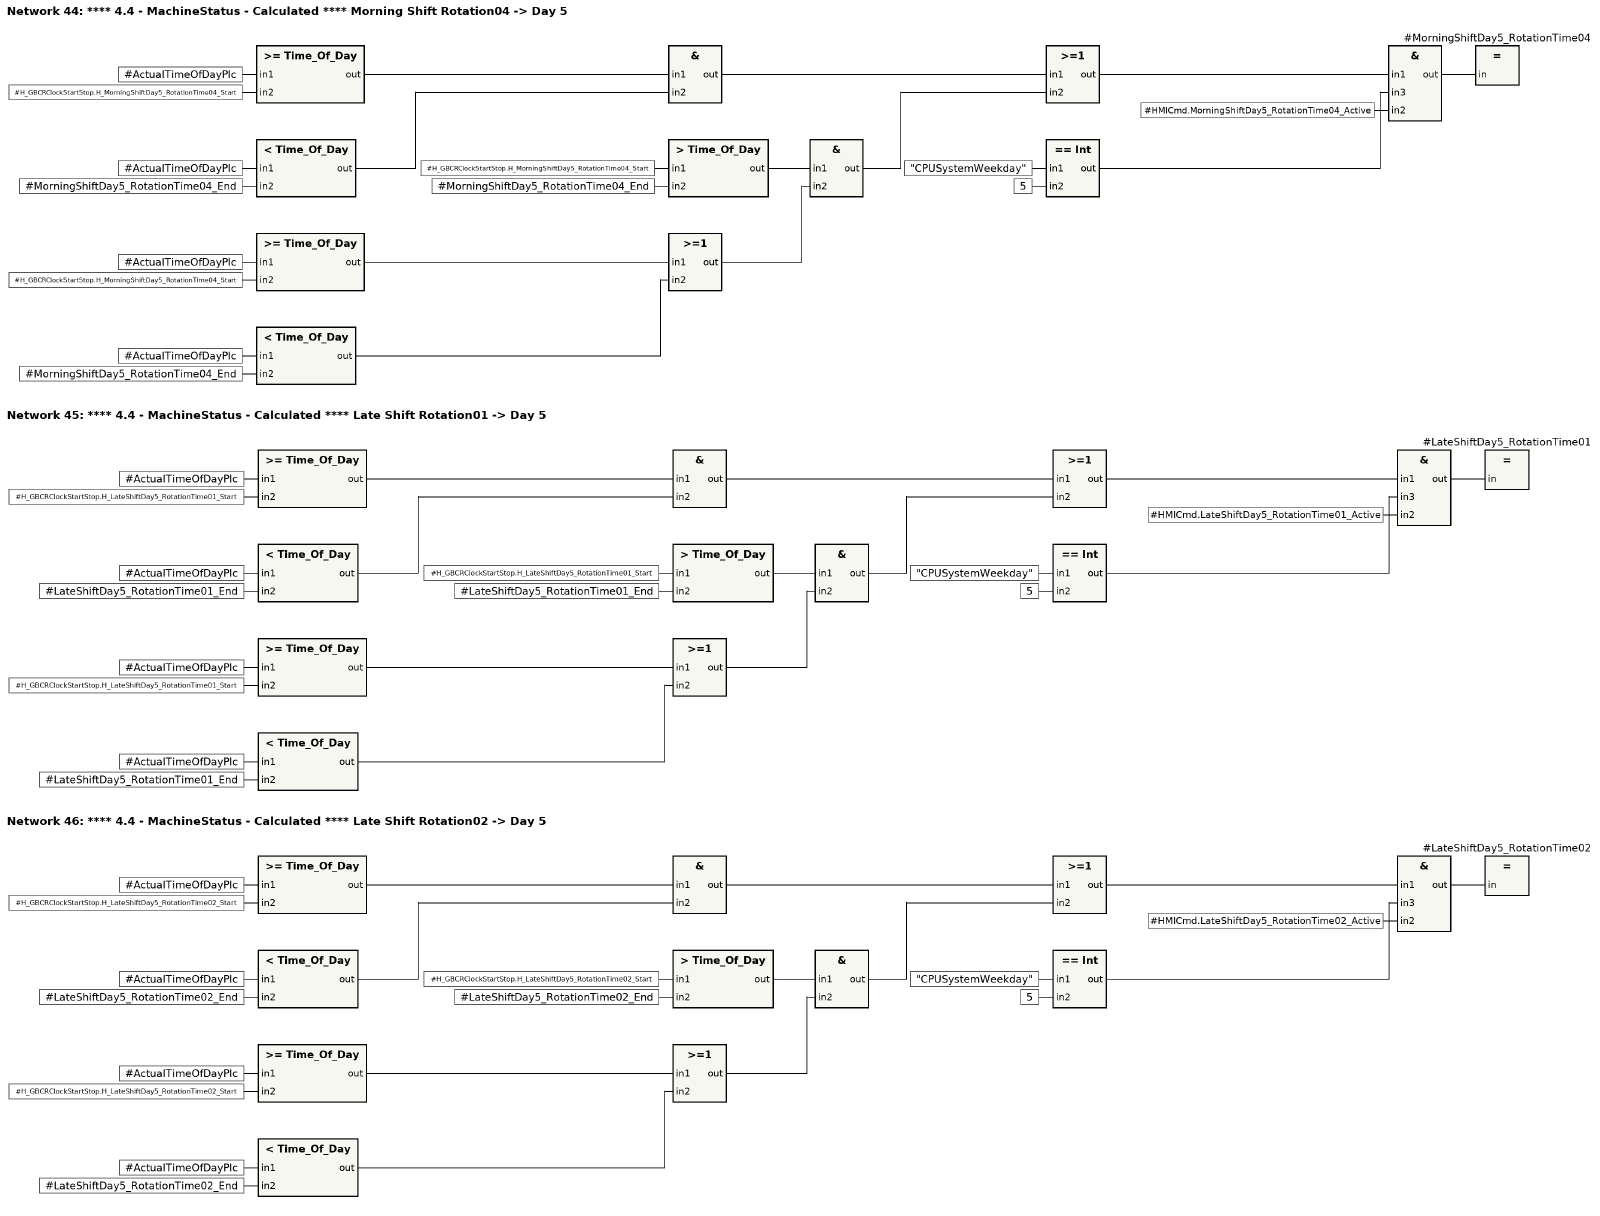
   #MorningShiftDay5_RotationTime04 := (((#ActualTimeOfDayPlc >= #H_GBCRClockStartStop.H_MorningShiftDay5_RotationTime04_Start) AND (#ActualTimeOfDayPlc < #MorningShiftDay5_RotationTime04_End)) OR ((#H_GBCRClockStartStop.H_MorningShiftDay5_RotationTime04_Start > #MorningShiftDay5_RotationTime04_End) AND ((#ActualTimeOfDayPlc >= #H_GBCRClockStartStop.H_MorningShiftDay5_RotationTime04_Start) OR (#ActualTimeOfDayPlc < #MorningShiftDay5_RotationTime04_End)))) AND ("CPUSystemWeekday" = 5) AND #HMICmd.MorningShiftDay5_RotationTime04_Active;
END_REGION

REGION Network 45: **** 4.4 - MachineStatus - Calculated **** Late Shift Rotation01 -> Day 5
   #LateShiftDay5_RotationTime01 := (((#ActualTimeOfDayPlc >= #H_GBCRClockStartStop.H_LateShiftDay5_RotationTime01_Start) AND (#ActualTimeOfDayPlc < #LateShiftDay5_RotationTime01_End)) OR ((#H_GBCRClockStartStop.H_LateShiftDay5_RotationTime01_Start > #LateShiftDay5_RotationTime01_End) AND ((#ActualTimeOfDayPlc >= #H_GBCRClockStartStop.H_LateShiftDay5_RotationTime01_Start) OR (#ActualTimeOfDayPlc < #LateShiftDay5_RotationTime01_End)))) AND ("CPUSystemWeekday" = 5) AND #HMICmd.LateShiftDay5_RotationTime01_Active;
END_REGION

REGION Network 46: **** 4.4 - MachineStatus - Calculated **** Late Shift Rotation02 -> Day 5
   #LateShiftDay5_RotationTime02 := (((#ActualTimeOfDayPlc >= #H_GBCRClockStartStop.H_LateShiftDay5_RotationTime02_Start) AND (#ActualTimeOfDayPlc < #LateShiftDay5_RotationTime02_End)) OR ((#H_GBCRClockStartStop.H_LateShiftDay5_RotationTime02_Start > #LateShiftDay5_RotationTime02_End) AND ((#ActualTimeOfDayPlc >= #H_GBCRClockStartStop.H_LateShiftDay5_RotationTime02_Start) OR (#ActualTimeOfDayPlc < #LateShiftDay5_RotationTime02_End)))) AND ("CPUSystemWeekday" = 5) AND #HMICmd.LateShiftDay5_RotationTime02_Active;
END_REGION

REGION Network 47: **** 4.4 - MachineStatus - Calculated **** Late Shift Rotation03 -> Day 5
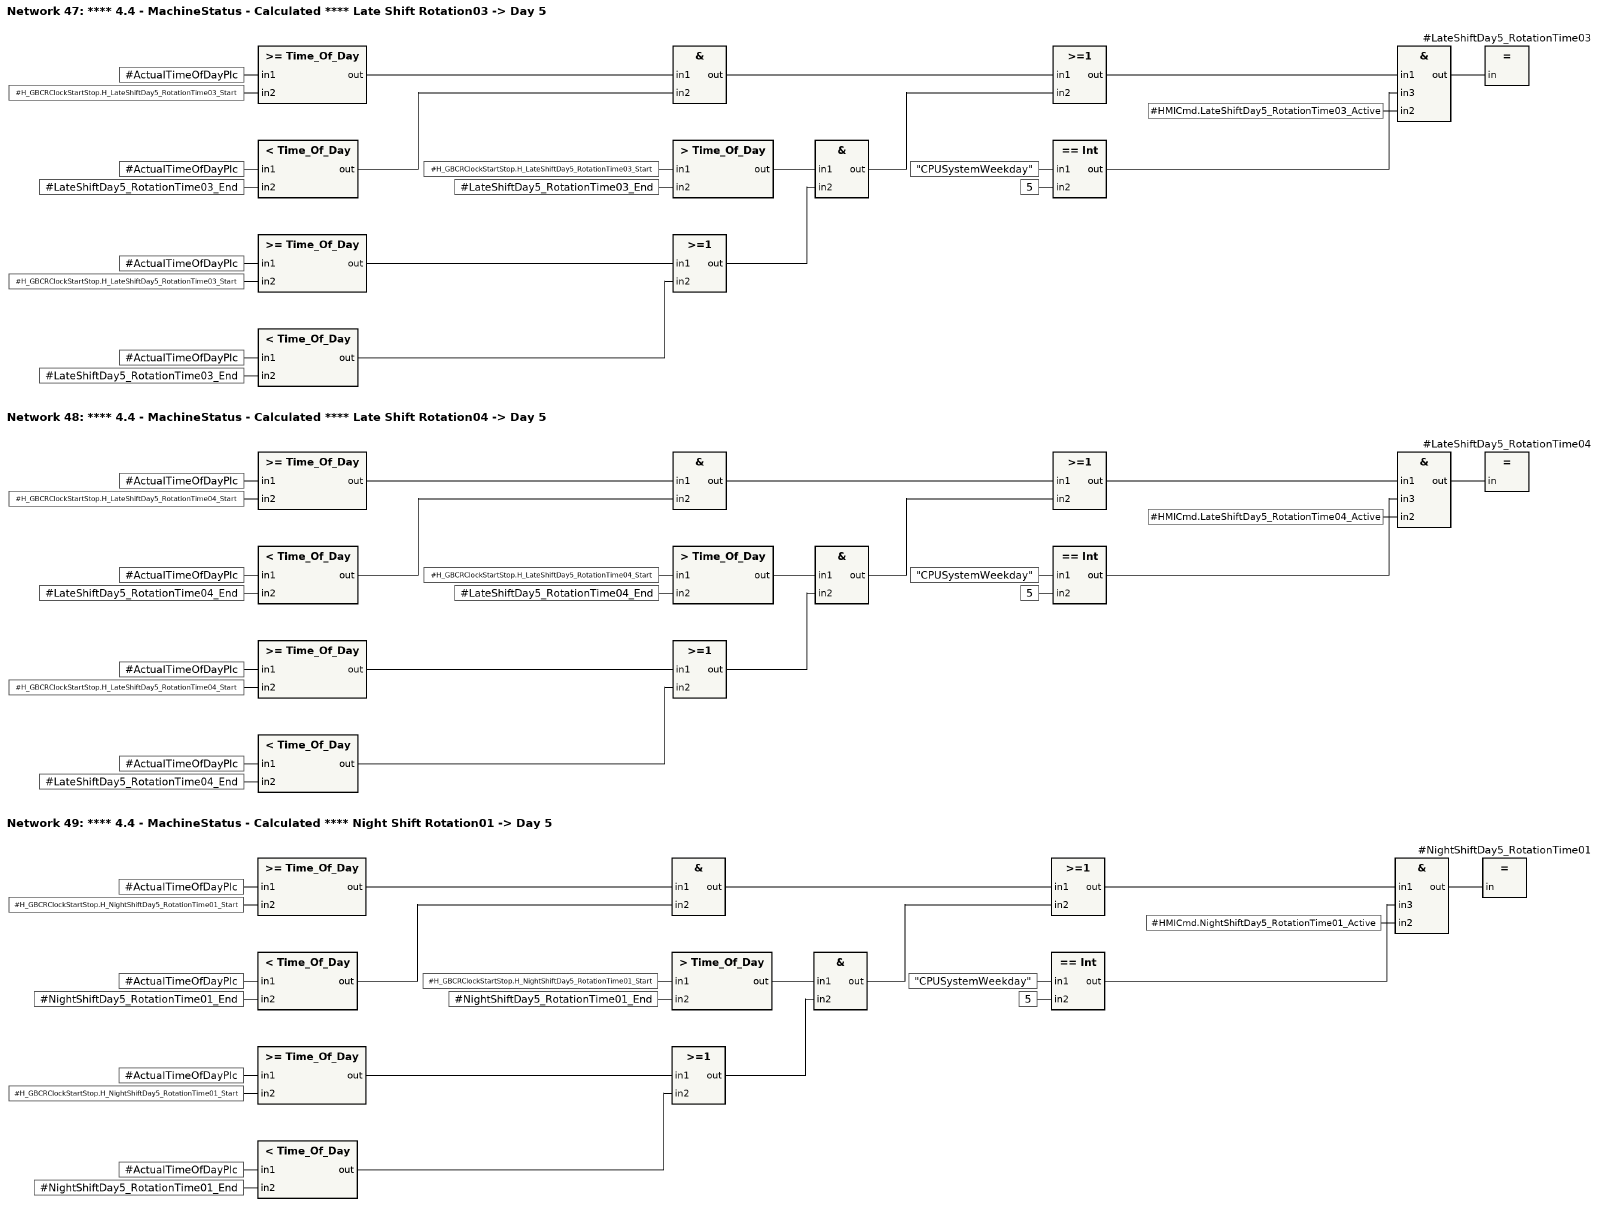
   #LateShiftDay5_RotationTime03 := (((#ActualTimeOfDayPlc >= #H_GBCRClockStartStop.H_LateShiftDay5_RotationTime03_Start) AND (#ActualTimeOfDayPlc < #LateShiftDay5_RotationTime03_End)) OR ((#H_GBCRClockStartStop.H_LateShiftDay5_RotationTime03_Start > #LateShiftDay5_RotationTime03_End) AND ((#ActualTimeOfDayPlc >= #H_GBCRClockStartStop.H_LateShiftDay5_RotationTime03_Start) OR (#ActualTimeOfDayPlc < #LateShiftDay5_RotationTime03_End)))) AND ("CPUSystemWeekday" = 5) AND #HMICmd.LateShiftDay5_RotationTime03_Active;
END_REGION

REGION Network 48: **** 4.4 - MachineStatus - Calculated **** Late Shift Rotation04 -> Day 5
   #LateShiftDay5_RotationTime04 := (((#ActualTimeOfDayPlc >= #H_GBCRClockStartStop.H_LateShiftDay5_RotationTime04_Start) AND (#ActualTimeOfDayPlc < #LateShiftDay5_RotationTime04_End)) OR ((#H_GBCRClockStartStop.H_LateShiftDay5_RotationTime04_Start > #LateShiftDay5_RotationTime04_End) AND ((#ActualTimeOfDayPlc >= #H_GBCRClockStartStop.H_LateShiftDay5_RotationTime04_Start) OR (#ActualTimeOfDayPlc < #LateShiftDay5_RotationTime04_End)))) AND ("CPUSystemWeekday" = 5) AND #HMICmd.LateShiftDay5_RotationTime04_Active;
END_REGION

REGION Network 49: **** 4.4 - MachineStatus - Calculated **** Night Shift Rotation01 -> Day 5
   #NightShiftDay5_RotationTime01 := (((#ActualTimeOfDayPlc >= #H_GBCRClockStartStop.H_NightShiftDay5_RotationTime01_Start) AND (#ActualTimeOfDayPlc < #NightShiftDay5_RotationTime01_End)) OR ((#H_GBCRClockStartStop.H_NightShiftDay5_RotationTime01_Start > #NightShiftDay5_RotationTime01_End) AND ((#ActualTimeOfDayPlc >= #H_GBCRClockStartStop.H_NightShiftDay5_RotationTime01_Start) OR (#ActualTimeOfDayPlc < #NightShiftDay5_RotationTime01_End)))) AND ("CPUSystemWeekday" = 5) AND #HMICmd.NightShiftDay5_RotationTime01_Active;
END_REGION

REGION Network 50: **** 4.4 - MachineStatus - Calculated **** Night Shift Rotation02 -> Day 5
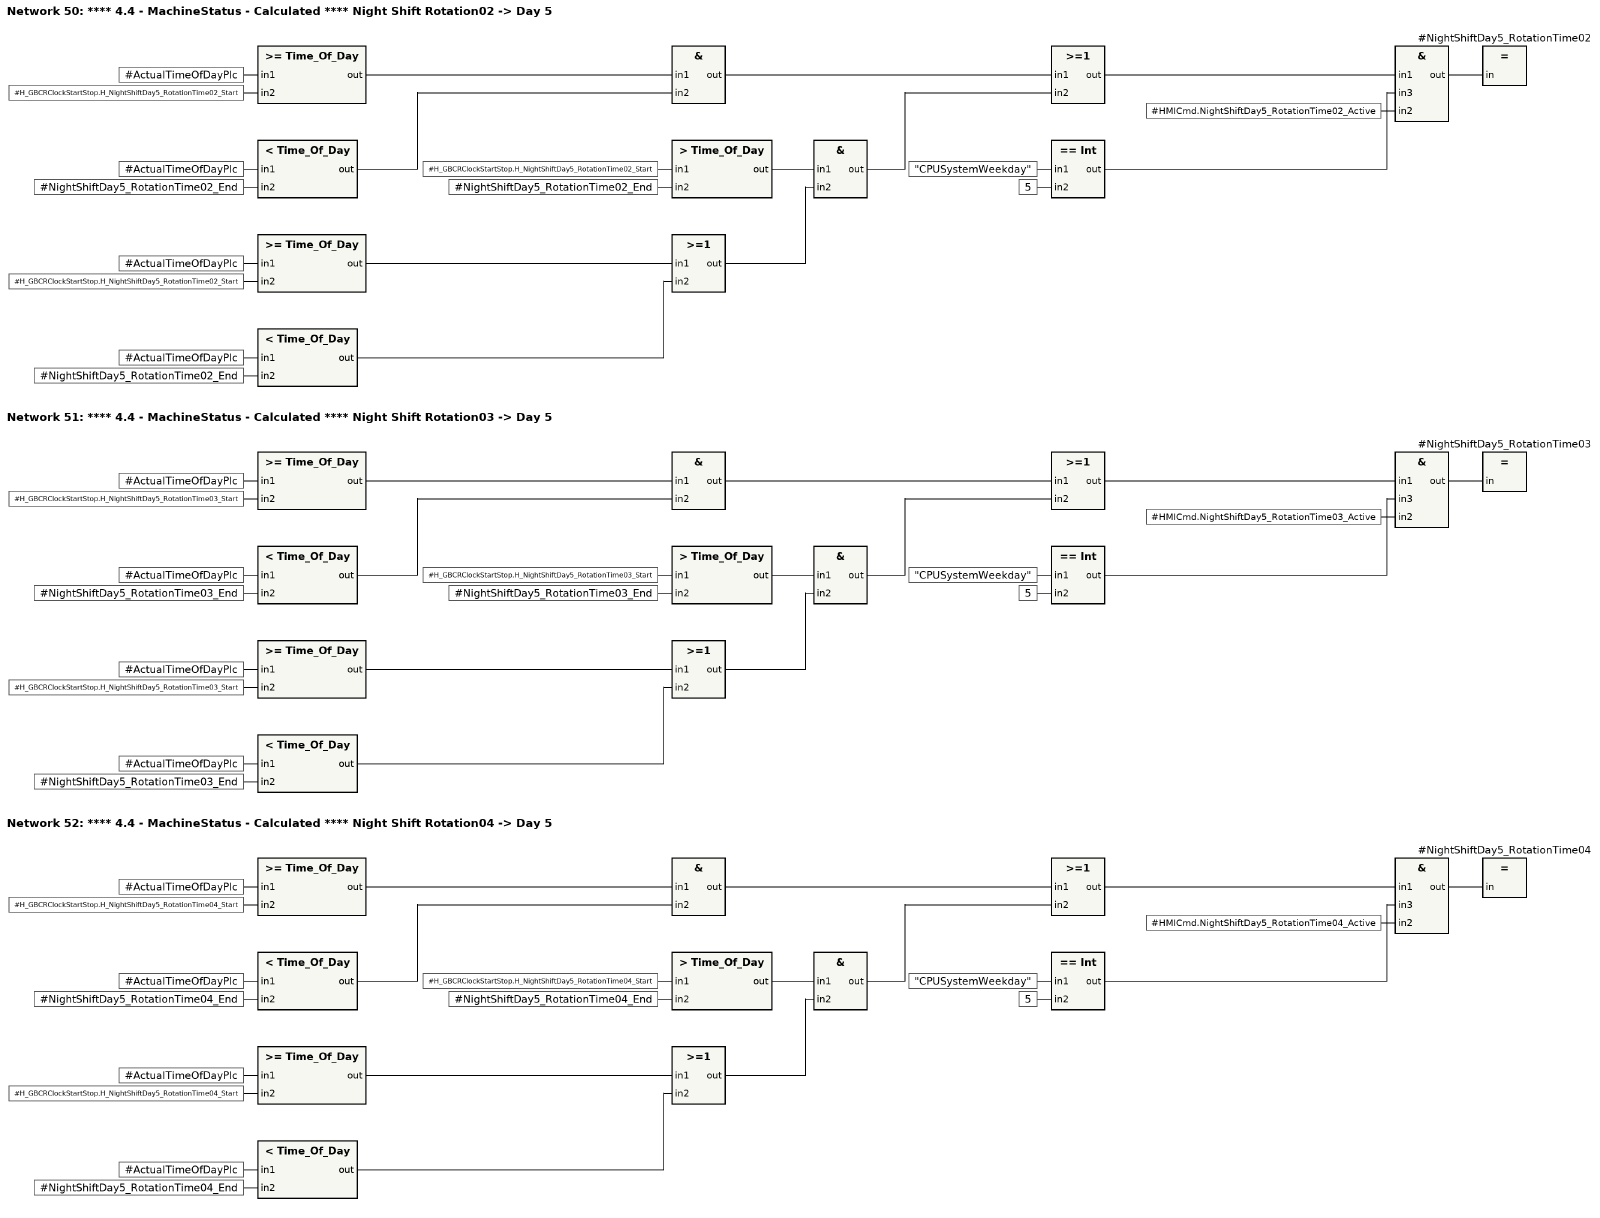
   #NightShiftDay5_RotationTime02 := (((#ActualTimeOfDayPlc >= #H_GBCRClockStartStop.H_NightShiftDay5_RotationTime02_Start) AND (#ActualTimeOfDayPlc < #NightShiftDay5_RotationTime02_End)) OR ((#H_GBCRClockStartStop.H_NightShiftDay5_RotationTime02_Start > #NightShiftDay5_RotationTime02_End) AND ((#ActualTimeOfDayPlc >= #H_GBCRClockStartStop.H_NightShiftDay5_RotationTime02_Start) OR (#ActualTimeOfDayPlc < #NightShiftDay5_RotationTime02_End)))) AND ("CPUSystemWeekday" = 5) AND #HMICmd.NightShiftDay5_RotationTime02_Active;
END_REGION

REGION Network 51: **** 4.4 - MachineStatus - Calculated **** Night Shift Rotation03 -> Day 5
   #NightShiftDay5_RotationTime03 := (((#ActualTimeOfDayPlc >= #H_GBCRClockStartStop.H_NightShiftDay5_RotationTime03_Start) AND (#ActualTimeOfDayPlc < #NightShiftDay5_RotationTime03_End)) OR ((#H_GBCRClockStartStop.H_NightShiftDay5_RotationTime03_Start > #NightShiftDay5_RotationTime03_End) AND ((#ActualTimeOfDayPlc >= #H_GBCRClockStartStop.H_NightShiftDay5_RotationTime03_Start) OR (#ActualTimeOfDayPlc < #NightShiftDay5_RotationTime03_End)))) AND ("CPUSystemWeekday" = 5) AND #HMICmd.NightShiftDay5_RotationTime03_Active;
END_REGION

REGION Network 52: **** 4.4 - MachineStatus - Calculated **** Night Shift Rotation04 -> Day 5
   #NightShiftDay5_RotationTime04 := (((#ActualTimeOfDayPlc >= #H_GBCRClockStartStop.H_NightShiftDay5_RotationTime04_Start) AND (#ActualTimeOfDayPlc < #NightShiftDay5_RotationTime04_End)) OR ((#H_GBCRClockStartStop.H_NightShiftDay5_RotationTime04_Start > #NightShiftDay5_RotationTime04_End) AND ((#ActualTimeOfDayPlc >= #H_GBCRClockStartStop.H_NightShiftDay5_RotationTime04_Start) OR (#ActualTimeOfDayPlc < #NightShiftDay5_RotationTime04_End)))) AND ("CPUSystemWeekday" = 5) AND #HMICmd.NightShiftDay5_RotationTime04_Active;
END_REGION

REGION Network 53: **** 4.6 - Machine status - Indications **** Icon Animation
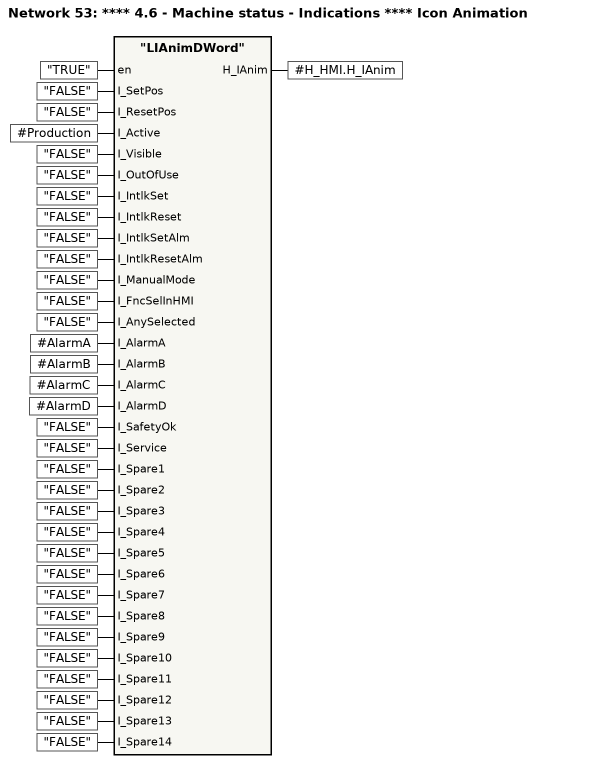
   IF "TRUE" THEN
       "LIAnimDWord"(I_SetPos := "FALSE",
                     I_ResetPos := "FALSE",
                     I_Active := #Production,
                     I_Visible := "FALSE",
                     I_OutOfUse := "FALSE",
                     I_IntlkSet := "FALSE",
                     I_IntlkReset := "FALSE",
                     I_IntlkSetAlm := "FALSE",
                     I_IntlkResetAlm := "FALSE",
                     I_ManualMode := "FALSE",
                     I_FncSelInHMI := "FALSE",
                     I_AnySelected := "FALSE",
                     I_AlarmA := #AlarmA,
                     I_AlarmB := #AlarmB,
                     I_AlarmC := #AlarmC,
                     I_AlarmD := #AlarmD,
                     I_SafetyOk := "FALSE",
                     I_Service := "FALSE",
                     I_Spare1 := "FALSE",
                     I_Spare2 := "FALSE",
                     I_Spare3 := "FALSE",
                     I_Spare4 := "FALSE",
                     I_Spare5 := "FALSE",
                     I_Spare6 := "FALSE",
                     I_Spare7 := "FALSE",
                     I_Spare8 := "FALSE",
                     I_Spare9 := "FALSE",
                     I_Spare10 := "FALSE",
                     I_Spare11 := "FALSE",
                     I_Spare12 := "FALSE",
                     I_Spare13 := "FALSE",
                     I_Spare14 := "FALSE",
                     H_IAnim => #H_HMI.H_IAnim);
   END_IF;
END_REGION

REGION Network 54: **** 4.6 - Machine status - Indications **** Animation
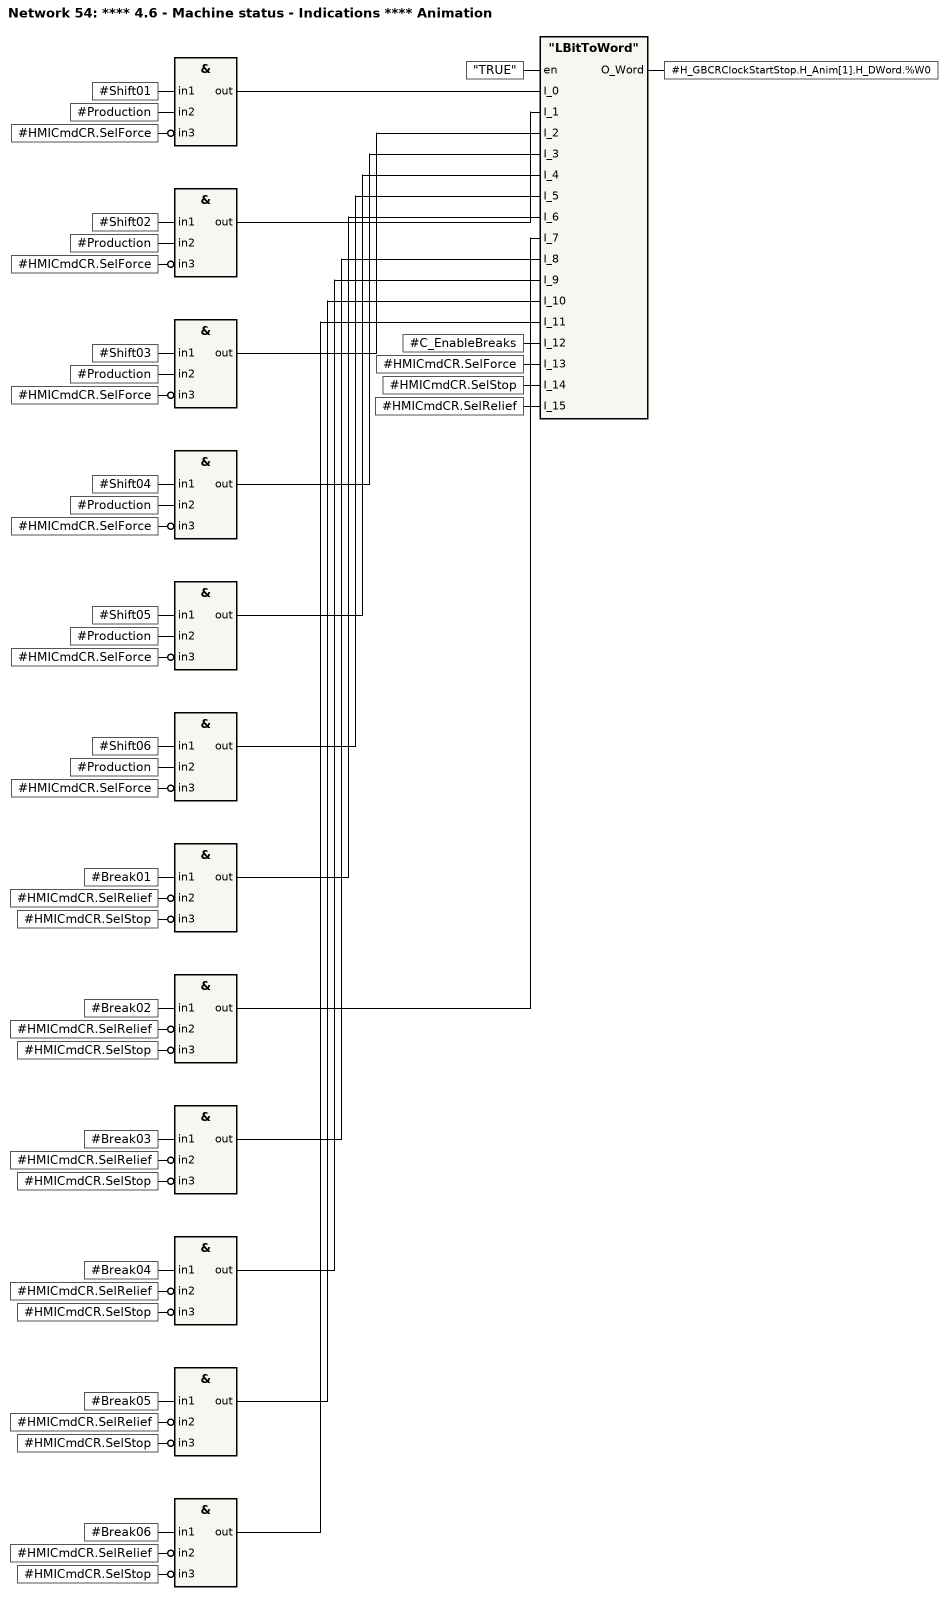
   IF "TRUE" THEN
       "LBitToWord"(I_0 := #Shift01 AND #Production AND NOT #HMICmdCR.SelForce,
                    I_1 := #Shift02 AND #Production AND NOT #HMICmdCR.SelForce,
                    I_2 := #Shift03 AND #Production AND NOT #HMICmdCR.SelForce,
                    I_3 := #Shift04 AND #Production AND NOT #HMICmdCR.SelForce,
                    I_4 := #Shift05 AND #Production AND NOT #HMICmdCR.SelForce,
                    I_5 := #Shift06 AND #Production AND NOT #HMICmdCR.SelForce,
                    I_6 := #Break01 AND NOT #HMICmdCR.SelRelief AND NOT #HMICmdCR.SelStop,
                    I_7 := #Break02 AND NOT #HMICmdCR.SelRelief AND NOT #HMICmdCR.SelStop,
                    I_8 := #Break03 AND NOT #HMICmdCR.SelRelief AND NOT #HMICmdCR.SelStop,
                    I_9 := #Break04 AND NOT #HMICmdCR.SelRelief AND NOT #HMICmdCR.SelStop,
                    I_10 := #Break05 AND NOT #HMICmdCR.SelRelief AND NOT #HMICmdCR.SelStop,
                    I_11 := #Break06 AND NOT #HMICmdCR.SelRelief AND NOT #HMICmdCR.SelStop,
                    I_12 := #C_EnableBreaks,
                    I_13 := #HMICmdCR.SelForce,
                    I_14 := #HMICmdCR.SelStop,
                    I_15 := #HMICmdCR.SelRelief,
                    O_Word => #H_GBCRClockStartStop.H_Anim[1].H_DWord.%W0);
   END_IF;
END_REGION

REGION Network 55: **** 4.6 - Machine status - Indications **** Animation2
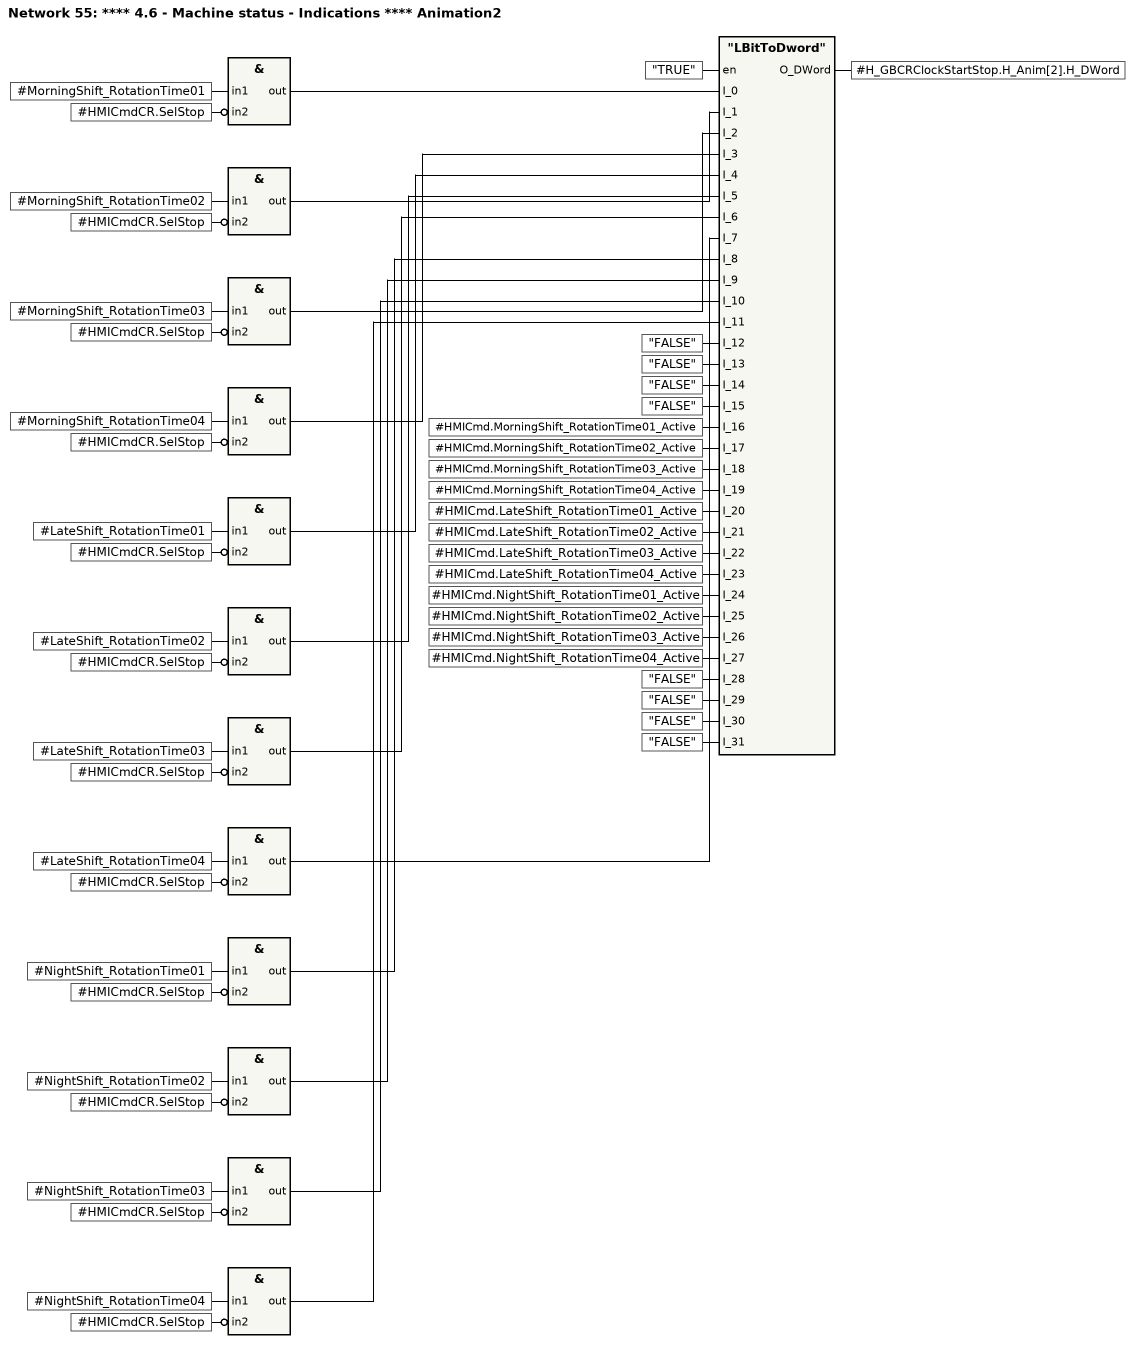
   IF "TRUE" THEN
       "LBitToDword"(I_0 := #MorningShift_RotationTime01 AND NOT #HMICmdCR.SelStop,
                     I_1 := #MorningShift_RotationTime02 AND NOT #HMICmdCR.SelStop,
                     I_2 := #MorningShift_RotationTime03 AND NOT #HMICmdCR.SelStop,
                     I_3 := #MorningShift_RotationTime04 AND NOT #HMICmdCR.SelStop,
                     I_4 := #LateShift_RotationTime01 AND NOT #HMICmdCR.SelStop,
                     I_5 := #LateShift_RotationTime02 AND NOT #HMICmdCR.SelStop,
                     I_6 := #LateShift_RotationTime03 AND NOT #HMICmdCR.SelStop,
                     I_7 := #LateShift_RotationTime04 AND NOT #HMICmdCR.SelStop,
                     I_8 := #NightShift_RotationTime01 AND NOT #HMICmdCR.SelStop,
                     I_9 := #NightShift_RotationTime02 AND NOT #HMICmdCR.SelStop,
                     I_10 := #NightShift_RotationTime03 AND NOT #HMICmdCR.SelStop,
                     I_11 := #NightShift_RotationTime04 AND NOT #HMICmdCR.SelStop,
                     I_12 := "FALSE",
                     I_13 := "FALSE",
                     I_14 := "FALSE",
                     I_15 := "FALSE",
                     I_16 := #HMICmd.MorningShift_RotationTime01_Active,
                     I_17 := #HMICmd.MorningShift_RotationTime02_Active,
                     I_18 := #HMICmd.MorningShift_RotationTime03_Active,
                     I_19 := #HMICmd.MorningShift_RotationTime04_Active,
                     I_20 := #HMICmd.LateShift_RotationTime01_Active,
                     I_21 := #HMICmd.LateShift_RotationTime02_Active,
                     I_22 := #HMICmd.LateShift_RotationTime03_Active,
                     I_23 := #HMICmd.LateShift_RotationTime04_Active,
                     I_24 := #HMICmd.NightShift_RotationTime01_Active,
                     I_25 := #HMICmd.NightShift_RotationTime02_Active,
                     I_26 := #HMICmd.NightShift_RotationTime03_Active,
                     I_27 := #HMICmd.NightShift_RotationTime04_Active,
                     I_28 := "FALSE",
                     I_29 := "FALSE",
                     I_30 := "FALSE",
                     I_31 := "FALSE",
                     O_DWord => #H_GBCRClockStartStop.H_Anim[2].H_DWord);
   END_IF;
END_REGION

REGION Network 56: **** 4.6 - Machine status - Indications **** Animation3
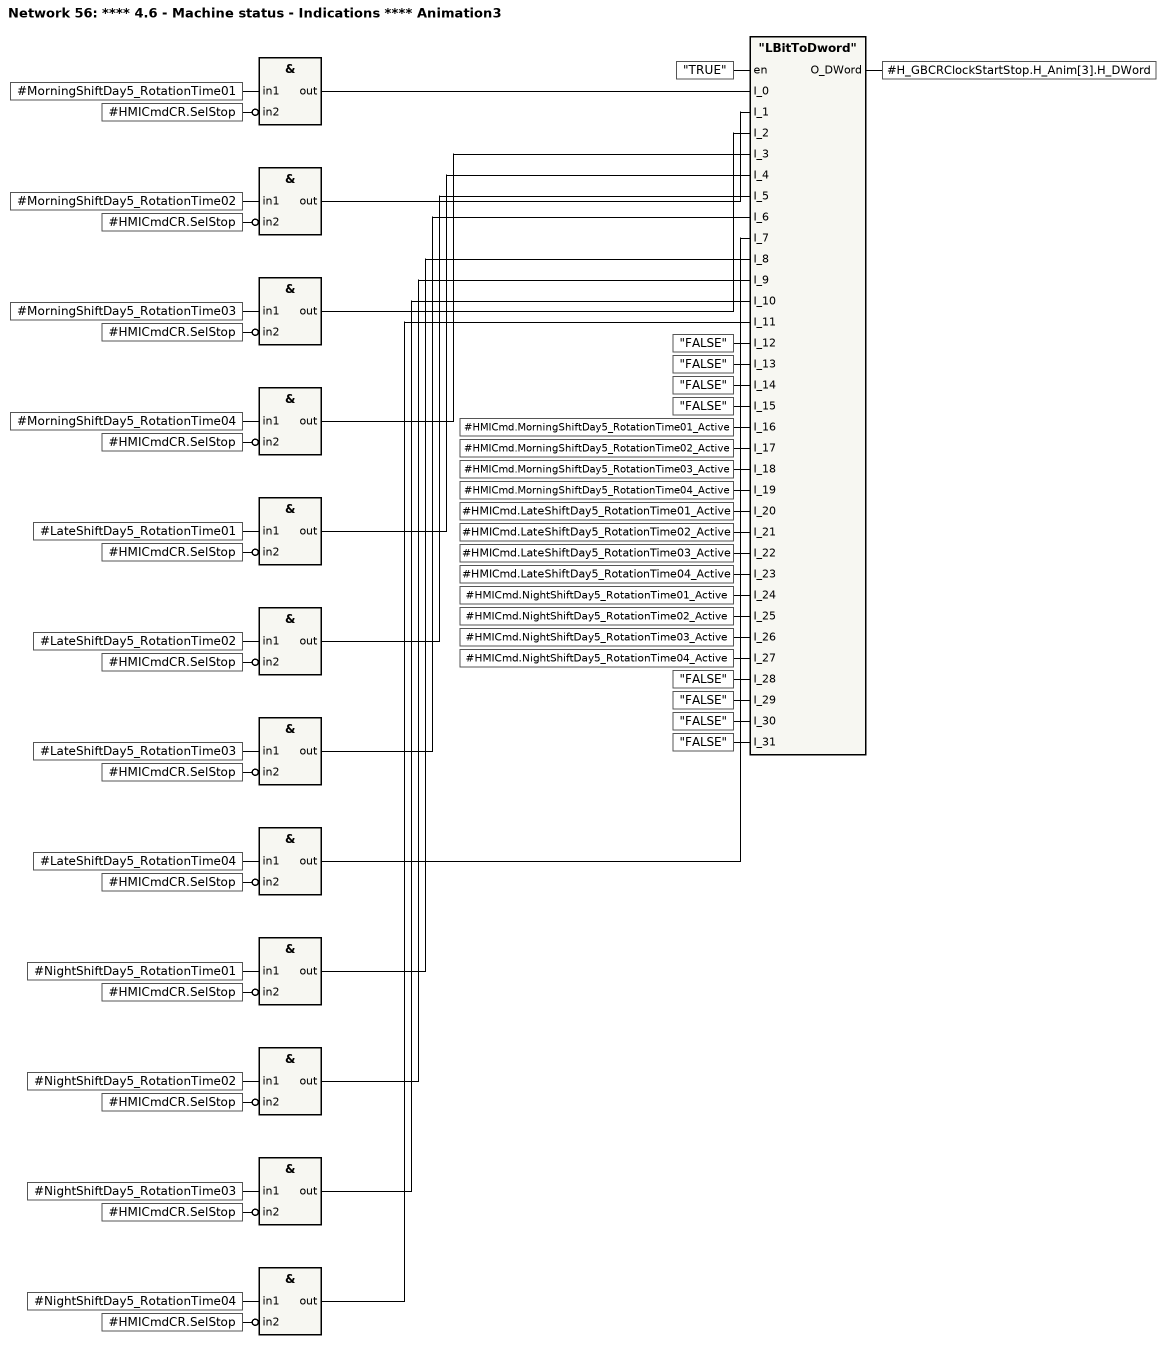
   IF "TRUE" THEN
       "LBitToDword"(I_0 := #MorningShiftDay5_RotationTime01 AND NOT #HMICmdCR.SelStop,
                     I_1 := #MorningShiftDay5_RotationTime02 AND NOT #HMICmdCR.SelStop,
                     I_2 := #MorningShiftDay5_RotationTime03 AND NOT #HMICmdCR.SelStop,
                     I_3 := #MorningShiftDay5_RotationTime04 AND NOT #HMICmdCR.SelStop,
                     I_4 := #LateShiftDay5_RotationTime01 AND NOT #HMICmdCR.SelStop,
                     I_5 := #LateShiftDay5_RotationTime02 AND NOT #HMICmdCR.SelStop,
                     I_6 := #LateShiftDay5_RotationTime03 AND NOT #HMICmdCR.SelStop,
                     I_7 := #LateShiftDay5_RotationTime04 AND NOT #HMICmdCR.SelStop,
                     I_8 := #NightShiftDay5_RotationTime01 AND NOT #HMICmdCR.SelStop,
                     I_9 := #NightShiftDay5_RotationTime02 AND NOT #HMICmdCR.SelStop,
                     I_10 := #NightShiftDay5_RotationTime03 AND NOT #HMICmdCR.SelStop,
                     I_11 := #NightShiftDay5_RotationTime04 AND NOT #HMICmdCR.SelStop,
                     I_12 := "FALSE",
                     I_13 := "FALSE",
                     I_14 := "FALSE",
                     I_15 := "FALSE",
                     I_16 := #HMICmd.MorningShiftDay5_RotationTime01_Active,
                     I_17 := #HMICmd.MorningShiftDay5_RotationTime02_Active,
                     I_18 := #HMICmd.MorningShiftDay5_RotationTime03_Active,
                     I_19 := #HMICmd.MorningShiftDay5_RotationTime04_Active,
                     I_20 := #HMICmd.LateShiftDay5_RotationTime01_Active,
                     I_21 := #HMICmd.LateShiftDay5_RotationTime02_Active,
                     I_22 := #HMICmd.LateShiftDay5_RotationTime03_Active,
                     I_23 := #HMICmd.LateShiftDay5_RotationTime04_Active,
                     I_24 := #HMICmd.NightShiftDay5_RotationTime01_Active,
                     I_25 := #HMICmd.NightShiftDay5_RotationTime02_Active,
                     I_26 := #HMICmd.NightShiftDay5_RotationTime03_Active,
                     I_27 := #HMICmd.NightShiftDay5_RotationTime04_Active,
                     I_28 := "FALSE",
                     I_29 := "FALSE",
                     I_30 := "FALSE",
                     I_31 := "FALSE",
                     O_DWord => #H_GBCRClockStartStop.H_Anim[3].H_DWord);
   END_IF;
END_REGION

REGION Network 57: **** 4.6 - Machine status - Indications **** Animation Shift Times
